// TwinCAT 3 PLC project Testlibrary
// Title: TestFramework
// Company: Hoox.Software
// Author: Patrick Dressel
// ProjectVersion: 2.2.6
// ProgramVersion: 3.1.4022.6
// libraries:
//   Tc2_Standard, * (Beckhoff Automation GmbH)
//   Tc2_System, * (Beckhoff Automation GmbH)
//   Tc2_Utilities, * (Beckhoff Automation GmbH)
//   Tc3_Module, * (Beckhoff Automation GmbH)
//   Base Interfaces,newest,System
// project tree:
//   Datatypes/ EResult_t.TcDUT, EAssertion_t.TcDUT (not stored), ERetCode_t.TcDUT (not stored), EState_t.TcDUT, IdHandle_t.TcDUT (not stored), ObjectId_t.TcDUT (not stored), SStatistic_t.TcDUT (not stored), STestcase_t.TcDUT, StringHandle_t.TcDUT (not stored), StrMessage_t.TcDUT (not stored), TestCaseHandle_t.TcDUT (not stored)
//   Datatypes/Report/ EExportState_t.TcDUT, EReportType_t.TcDUT (not stored), NameHandle_t.TcDUT (not stored), PathHandle_t.TcDUT (not stored), StrFileName_t.TcDUT (not stored), StrPathName_t.TcDUT (not stored), TestReportHandle_t.TcDUT (not stored), UBaseTypes_t.TcDUT (not stored), UTime_t.TcDUT (not stored)
//   GVLs/ GVL_Sample.TcGVL (excluded from build)
//   / GVL_Parameter.TcGVL, PlcTask.TcTTO
//   Source/Report/File/ FB_CoverageFile.TcPOU, FB_FileBase.TcPOU, FB_TestReportBase.TcPOU, FB_TextReport.TcPOU, IFileData_t.TcIO
//   Source/Report/Format/ EXmlFormat_t.TcDUT, FB_XmlTag.TcPOU, _CONCAT.TcPOU, _LEN.TcPOU
//   Source/Testlib/ FB_Assertion.TcPOU (not stored), PRG_TestLib.TcPOU
//   Source/Testsuite/ FB_Testsuite.TcPOU, ITestsuite_t.TcIO
//   Source/TestBase/ FB_TestBase.TcPOU (not stored), ITestBase_t.TcIO
//   Test/ FB_Test_Base.TcPOU, FB_Test_Base_Ptr.TcPOU, FB_Test_Base_Not.TcPOU, FB_Test_Base_Delay.TcPOU, PRG_Temp.TcPOU
// real-time tasks:
//   TASK PlcTask: cycle T#10ms, priority 20, ADS port 350

CONFIGURATION Testlibrary
    RESOURCE PLC ON TwinCAT3
        TASK PlcTask(INTERVAL := T#10ms, PRIORITY := 20);
        PROGRAM PRG_TestLib WITH PlcTask : PRG_TestLib;
        PROGRAM PRG_Temp WITH PlcTask : PRG_Temp;
    END_RESOURCE
END_CONFIGURATION

// ---- Datatypes/EResult_t.TcDUT
{attribute 'qualified_only'}
{attribute 'strict'}
TYPE EResult_t :
(
   eStateIdle,
	eStateSkipped,
	eStatePassed,
	eStateFailed,
	eStateFailedFatal
);
END_TYPE

// ---- Datatypes/EState_t.TcDUT
{attribute 'qualified_only'}
{attribute 'strict'}
TYPE EState_t :
(
	eStateInit,
	eStateIdle,
	eStatePrepare,
	eStateExecute,
	eStateCleanUp,
	eStateBuildUnitTestFile,
	eStateReady,
	eStateExport,
	eStateError,
	eStateLicenseError
);
END_TYPE

// ---- Datatypes/Report/EExportState_t.TcDUT
{attribute 'qualified_only'}
{attribute 'strict'}
TYPE EExportState_t :
(
	eExportIdle := 0,
	eExportOpen,
	eExportGetLine,
	eExportWrite,
	eExportClose,
	eExportError
);
END_TYPE

// ---- Datatypes/STestcase_t.TcDUT
TYPE STestcase_t :
STRUCT
	u32Passed 		: UDINT;
	u32Failed 		: UDINT;
	u32Time         : UDINT;
	eState          : EResult_t;
END_STRUCT
END_TYPE

// ---- Source/Report/Format/EXmlFormat_t.TcDUT
{attribute 'qualified_only'}
{attribute 'strict'}
TYPE EXmlFormat_t :
(
	ePlainXml := 0,
	eStructuredXml
);
END_TYPE

// ---- GVLs/GVL_Sample.TcGVL
{attribute 'qualified_only'}
VAR_GLOBAL
	// This File is only a simple Demo to show the usage of the Library
    // Using the Sccx-Script it can be generated by a build server like Jenkins

	// Report Instance 
	fb_TestReport : FB_TextReport;	
	
	// Register Testsuite
    // Testuite connects itself to PRG_TestLib
	fb_TestSuite1 : FB_Testsuite(i_strId 	:= 'TestSuite1', 	
								 i_strPath	:= 'Testframework\Testframework\UnitTest\');
	
	// Register Test in Testsuite1
    // Testcase connect itself to given Testsuite interface
    // set Execute to false to skip the test.
	fb_Test   : FB_Test_Base( i_strId 	 	    := 'TF1.1',
                              i_strClassName	:= 'FB_TestBase.TcPOU',
                              i_strPath 		:= 'Source',
                              i_iTestSuite 	    := fb_TestSuite1,
                              i_bExecute   	    := TRUE);
										
	fb_Test2   : FB_Test_Base( i_strId 	 	    := 'TF2.1',
                              i_strClassName	:= 'FB_TestBase.TcPOU',
                              i_strPath 		:= 'Source',
                              i_iTestSuite 	    := fb_TestSuite1,
                              i_bExecute   	    := TRUE);										
END_VAR

// ---- GVL_Parameter.TcGVL
{attribute 'qualified_only'}
VAR_GLOBAL CONSTANT
	strExportDirectory : STRING := 'C:\testresult\';
END_VAR

// ---- Source/Report/File/IFileData_t.TcIO
INTERFACE IFileData_t

METHOD getDataPtr : POINTER TO BYTE
END_METHOD

METHOD getSize : UDINT
VAR_INPUT
END_VAR
END_METHOD

END_INTERFACE

// ---- Source/Testsuite/ITestsuite_t.TcIO
INTERFACE ITestsuite_t

METHOD PUBLIC addTestcase : BOOL
VAR_INPUT
	i_iTestCase : ITestBase_t;
END_VAR
END_METHOD

METHOD execute : BOOL
VAR_INPUT
    i_bStart : BOOL;
END_VAR
END_METHOD

METHOD getFirstTestCase : ITestBase_t
VAR_INPUT
END_VAR
END_METHOD

METHOD getId : STRING
VAR_INPUT
END_VAR
END_METHOD

METHOD getNextTestCase : ITestBase_t
VAR_INPUT
END_VAR
END_METHOD

METHOD getPath : ObjectId_t
VAR_INPUT
END_VAR
END_METHOD

METHOD getResult : EResult_t
VAR_INPUT
END_VAR
END_METHOD

METHOD getState : EState_t
VAR_INPUT
END_VAR
END_METHOD

PROPERTY Result : SStatistic_t
GET
END_GET
END_PROPERTY

END_INTERFACE

// ---- Source/TestBase/ITestBase_t.TcIO
INTERFACE ITestBase_t

METHOD PUBLIC FINAL _cleanup : ERetCode_t
VAR_INPUT
END_VAR
END_METHOD

METHOD PUBLIC FINAL _execute : ERetCode_t
VAR_INPUT
END_VAR
END_METHOD

METHOD PUBLIC FINAL _prepare : ERetCode_t
VAR_INPUT
END_VAR
END_METHOD

METHOD getClassname : ObjectId_t
VAR_INPUT
END_VAR
END_METHOD

METHOD getId : ObjectId_t
VAR_INPUT
END_VAR
END_METHOD

METHOD getMessage : StrMessage_t
VAR_INPUT
END_VAR
END_METHOD

METHOD getPath : ObjectId_t
VAR_INPUT
END_VAR
END_METHOD

PROPERTY Result : STestcase_t
GET
END_GET
END_PROPERTY

END_INTERFACE

// ---- Source/Testlib/PRG_TestLib.TcPOU
(******************************************************************************
Baustein: PRG_TestLibrary
Spezifikation: doc/Spezifikation.pdf, Kap. x.y.z
-------------------------------------------------------------------------------
erstellt:
von:
Geändert:
von:
-------------------------------------------------------------------------------
Beschreibung
Dieser Baustein etnhält alle Testsuites und führt diese aus.

-------------------------------------------------------------------------------
Input
	i_bStart : mit positiver Flanke werden die registrierten Testsuites ausgeführt

Output
	o_eState  		: EState_t;
	o_eResult 		: EResult_t;
	o_sStatistic	: SStatistic_t;
******************************************************************************)
{attribute 'global_init_slot' := '41000'}
PROGRAM PRG_TestLib
VAR_INPUT
	i_bStart : BOOL;
END_VAR
VAR_OUTPUT
	o_eState  		: EState_t;
	o_eResult 		: EResult_t;
	o_sStatistic	: SStatistic_t;
END_VAR
VAR
	bHwStart AT %I* : BOOL;
	bHwBusy  AT %Q* : BOOL;
	bHwReady AT %Q* : BOOL;
	
	a_iTestSuite 	: ARRAY [0..255] OF ITestSuite_t;
	u16TestSuites 	: UINT;
	u16Index	  		: UINT;
	iActTestSuite 	: ITestSuite_t;
	pTestReport		: POINTER TO FB_TestReportBase;
	eRetCode 		: ERetCode_t;

	fbSystemTime 		: FB_LocalSystemTime;
	
	fbExportFolder		: FB_CreateDir;
	fbUnittest 			: FB_CoverageFile;
	u16ReportState  	: UINT;
	u16TestSuitIdx		: UINT;
	iTestCase  			: ITestBase_t;
	sTempResult     	: SStatistic_t;
	
	xmlTestsuites	  	: FB_XmlTag;
	xmlTestsuite	  	: FB_XmlTag;
	xmlTest	  			: FB_XmlTag;
	xmlTestResult		: FB_XmlTag;		
END_VAR
VAR CONSTANT 
	ADSERR_DEVICE_ACCESSDENIED : UDINT := 16#723;
	ADSERR_DEVICE_NOTFOUND     : UDINT := 16#70C;
	ADSERR_DEVICE_EXISTS     	: UDINT := 16#70F;
END_VAR


	fbSystemTime(bEnable := TRUE, dwCycle := 5);
			
	fbUnittest();

	CASE o_eState OF 
	
	EState_t.eStateInit:	
		
		IF checkExportFolder() THEN 
		   logInfo('Testlib V2.2.6 Ready');
			o_eState := EState_t.eStateIdle; 
		END_IF

	EState_t.eStateIdle:
	
		IF i_bStart = TRUE OR bHwStart = TRUE THEN
			logInfo('+++++++++++++ Testbeginn ++++++++++++++');
			o_eState := EState_t.eStatePrepare;
			bHwReady := FALSE;
		END_IF
	
	EState_t.eStatePrepare:
	
		bHwBusy := TRUE;
		
		o_eResult 	  					:= EResult_t.eStatePassed;
		o_sStatistic.u32Executed 	:= 0;
		o_sStatistic.u32TestCases	:= 0;
		o_sStatistic.u32Asserts  	:= 0;
		o_sStatistic.u32Passed   	:= 0;
		o_sStatistic.u32Failed	 	:= 0;	

		iActTestSuite := getFirstTestSuite();
		
		IF iActTestSuite      <> 0   THEN
			o_eState := EState_t.eStateExecute;
		ELSE
			o_eState := EState_t.eStateError;	
		END_IF
	
	EState_t.eStateExecute:
	
		iActTestSuite.execute(i_bStart := TRUE);
	
		IF iActTestSuite.getState() = EState_t.eStateReady THEN
			
			IF iActTestSuite.getResult() = EResult_t.eStateFailed THEN
				o_eResult := EResult_t.eStateFailed;
			END_IF
			
			iActTestSuite.execute(i_bStart := FALSE);
			sTempResult := iActTestSuite.Result;

			o_eState := EState_t.eStateCleanUp;

			o_sStatistic.u32Executed 	:= o_sStatistic.u32Executed  + sTempResult.u32Executed;
			o_sStatistic.u32TestCases	:= o_sStatistic.u32TestCases + sTempResult.u32TestCases; 
			o_sStatistic.u32Asserts  	:= o_sStatistic.u32Asserts   + sTempResult.u32Asserts;
			o_sStatistic.u32Passed   	:= o_sStatistic.u32Passed    + sTempResult.u32Passed;
			o_sStatistic.u32Failed	 	:= o_sStatistic.u32Failed    + sTempResult.u32Failed;
		END_IF
	
	EState_t.eStateCleanUp:
	
		IF iActTestSuite.getResult() = EResult_t.eStateFailedFatal THEN
			o_eResult := EResult_t.eStateFailedFatal;
			o_eState  := EState_t.eStateExport;
			logInfo('+++++++++++++ Fatal Error : Test Ende ++++++++++++++');
		ELSE
			
			iActTestSuite := getNextTestSuite();
						
			IF iActTestSuite <> 0 THEN
				o_eState := EState_t.eStateExecute;
			ELSE
				o_eState := EState_t.eStateBuildUnitTestFile;
				logInfo('+++++++++++++ Test Ende ++++++++++++++');
			END_IF		
			
		END_IF

	EState_t.eStateExport:

		IF createReport(EReporttype_t.eExternalReport) = ERetCode_t.eRetDone THEN
			o_eState := EState_t.eStateBuildUnitTestFile;
		END_IF;
		
	EState_t.eStateBuildUnitTestFile:

		IF createReportnew(EReporttype_t.eUnitTestReport) = ERetCode_t.eRetDone THEN
			o_eState := EState_t.eStateReady;
		END_IF;
		
	EState_t.eStateReady:

		bHwReady := TRUE;
		bHwBusy  := FALSE;
		IF i_bStart  = FALSE AND 
			bHwStart = FALSE THEN
			o_eState := EState_t.eStateIdle;
		END_IF		
		
	EState_t.eStateError,
	EState_t.eStateLicenseError:
	
		bHwBusy  := FALSE;
		o_eState := EState_t.eStateError;

	END_CASE

(******************************************************************************
Baustein: PRG_UnitTestLib.addTestReport
Spezifikation: doc/Spezifikation.pdf, Kap. x.y.z
-------------------------------------------------------------------------------
erstellt:
von:
Geändert:
von:
-------------------------------------------------------------------------------
Beschreibung
Diese Methode

-------------------------------------------------------------------------------
Input
i_pTestReport

Output
-
******************************************************************************)
{attribute 'hide'} 
METHOD PUBLIC addTestReport : BOOL
VAR_INPUT
	i_pTestReport : TestReportHandle_t;
END_VAR

	pTestReport := i_pTestReport;
END_METHOD

(******************************************************************************
Baustein: PRG_UnitTestLib.addTestSuite
Spezifikation: doc/Spezifikation.pdf, Kap. x.y.z
-------------------------------------------------------------------------------
erstellt:
von:
Geändert:
von:
-------------------------------------------------------------------------------
Beschreibung
Diese Methode

-------------------------------------------------------------------------------
Input
i_pTestSuite

Output
-
******************************************************************************)
{attribute 'hide'} 
METHOD PUBLIC addTestSuite : BOOL
VAR_INPUT
	i_iTestSuite : ITestSuite_t;
END_VAR
VAR
    sStatistic : SStatistic_t;
END_VAR

	addTestSuite := FALSE;

	IF 	i_iTestSuite  <> 0   AND 
		u16TestSuites <  255 THEN
		
		a_iTestSuite[u16TestSuites] := i_iTestSuite;
		sStatistic      := i_iTestSuite.Result;
		u16TestSuites   := u16TestSuites +1;
	
		o_sStatistic.u32TestSuites := o_sStatistic.u32TestSuites + 1;
		o_sStatistic.u32TestCases  := o_sStatistic.u32TestCases + sStatistic.u32TestCases;
		
		addTestSuite := TRUE;
	END_IF
END_METHOD

// 
// Lt. Infosys wird ADSERR_DEVICE_ACCESSDENIED zurückgegeben wenn der
// Ordner bereits existiert. Das reicht an der Stelle um zu wissen das 
// es soweit passt.
{attribute 'hide'} 
METHOD INTERNAL checkExportFolder : BOOL

	checkExportFolder := FALSE;
	
	fbExportFolder(sNetId 		:= '',
						sPathName 	:= GVL_Parameter.strExportDirectory,
						ePath 		:= E_OpenPath.PATH_GENERIC,
						bExecute 	:= TRUE,
						tTimeout 	:= T#5S);
						
	IF (fbExportFolder.bBusy  = FALSE) AND 
		(fbExportFolder.bError = FALSE OR 
			fbExportFolder.nErrId = ADSERR_DEVICE_ACCESSDENIED OR 
			fbExportFolder.nErrId = ADSERR_DEVICE_EXISTS 		OR 
			fbExportFolder.nErrId = ADSERR_DEVICE_NOTFOUND) THEN
		checkExportFolder := true;
	END_IF;
END_METHOD

{attribute 'hide'} 
METHOD PRIVATE createReport : ERetCode_t
VAR_INPUT
	i_eReporttype : EReportType_t;
END_VAR
VAR
	eRetcode    : ERetCode_t;
	u32Temp     : UDINT;
	sTestResult : STestcase_t;
	sStatistic  : SStatistic_t;
END_VAR

	createReport := ERetCode_t.eRetBusy;

	CASE u16ReportState OF

	0: 
		IF i_eReporttype = EReportType_t.eUnitTestReport THEN
			u16ReportState := 20;
		END_IF;

		IF i_eReporttype = EReportType_t.eExternalReport THEN
			u16ReportState := 100;
		END_IF;

// +++++++++++++++++++++++++++++++++++++++++++++++++++++++++++
//
// Export Unittest Ergebnisse
// 
// +++++++++++++++++++++++++++++++++++++++++++++++++++++++++++
	20:		

		eRetcode := fbUnitTest.open(GVL_Parameter.strExportDirectory, 'Unittest.xml');

		IF eRetcode = ERetCode_t.eRetDone THEN

			u16ReportState := 21;

		ELSIF eRetcode = ERetCode_t.eRetFailed THEN

			logError('createReport Unittest.xml : Datei nicht geöffnet');
			u16ReportState := 22;

		END_IF;	

	21:

		u16TestSuitIdx := 0;

		fbUnitTest.addString('<?xml version="1.0" ?>');
		fbUnitTest.addCrlf();

		iActTestSuite := getFirstTestSuite();
		fbUnitTest.addString('<testsuites>');
		fbUnitTest.addCrlf();

		WHILE (iActTestSuite <> 0) DO

            sStatistic := iActTestSuite.Result;
			u16TestSuitIdx := u16TestSuitIdx+1;

			fbUnitTest.addString('<testsuite');
			fbUnitTest.addString(' name="');
			fbUnitTest.addString(iActTestSuite.getId());
			fbUnitTest.addString('" tests="');			
			fbUnitTest.addValue(sStatistic.u32TestCases);
			fbUnitTest.addString('" disabled="');
            u32Temp := sStatistic.u32TestCases-sStatistic.u32Executed;
			fbUnitTest.addValue(u32Temp);
			fbUnitTest.addString('" errors="');
			fbUnitTest.addValue(u32Temp);
			fbUnitTest.addString('" failures="');
			fbUnitTest.addValue(sStatistic.u32Failed);
			fbUnitTest.addString('" hostname="');
			fbUnitTest.addString('" id="');
			fbUnitTest.addvalue(u16TestSuitIdx);
			fbUnitTest.addString('" package="');
			fbUnitTest.addString(iActTestSuite.getPath());
			fbUnitTest.addString('">');
			fbUnitTest.addCrlf();

			iTestCase := iActTestSuite.getFirstTestCase();

			WHILE (iTestCase <> 0) DO
        
                sTestResult := iTestCase.Result;

				fbUnitTest.addString('<testcase');
				fbUnitTest.addString(' name="');
				fbUnitTest.addString(iTestCase.getId());
				fbUnitTest.addString('" assertions="');
                u32Temp := sTestResult.u32Failed + sTestResult.u32Passed;
				fbUnitTest.addValue(u32Temp);
				fbUnitTest.addString('" classname="');
				fbUnitTest.addString(iTestCase.getPath());
                fbUnitTest.addString('.');
				fbUnitTest.addString(iTestCase.getClassName());
				fbUnitTest.addString('" time="');				
				fbUnitTest.addTimeMs(sTestResult.u32Time);
				fbUnitTest.addString('">');
				fbUnitTest.addCrlf();

				CASE sTestResult.eState OF

				EResult_t.eStatePassed :

					fbUnitTest.addString('<passed/>');

				EResult_t.eStateFailed, 
				EResult_t.eStateFailedFatal :
			
					fbUnitTest.addString('<failure');
					fbUnitTest.addString(' message="');
					fbUnitTest.addString(iTestCase.getMessage());
					fbUnitTest.addString('"/>');
					
				EResult_t.eStateSkipped:

					fbUnitTest.addString('<skipped/>');

				END_CASE;
				
				fbUnitTest.addCrlf();	

				fbUnitTest.addString('</testcase>');
				fbUnitTest.addCrlf();		

				iTestCase := iActTestSuite.getNextTestCase();
		
			END_WHILE

			fbUnitTest.addString('</testsuite>');
			fbUnitTest.addCrlf();	

			iActTestSuite := getNextTestSuite();

		END_WHILE

		fbUnitTest.addString('</testsuites>');
		fbUnitTest.addCrlf();

		u16ReportState := 22;

	22:
		IF fbUnitTest.o_bOpen  = TRUE AND 
		   fbUnitTest.o_bEmpty = TRUE THEN
			fbUnitTest.close();
		END_IF;

		IF fbUnitTest.o_bOpen  = FALSE THEN
			createReport 	:= ERetCode_t.eRetDone;
		END_IF;

// +++++++++++++++++++++++++++++++++++++++++++++++++++++++++++
//
//
// 
// +++++++++++++++++++++++++++++++++++++++++++++++++++++++++++
	100:

		IF pTestReport <> 0 THEN
			
			createReport := pTestReport^.create();		
			
		ELSE

			createReport := ERetCode_t.eRetDone;

		END_IF;

	ELSE
		createReport := ERetCode_t.eRetFailed;
	END_CASE;

	IF createReport = ERetCode_t.eRetDone THEN
		u16ReportState := 0;
	END_IF;
















(**)
END_METHOD

{attribute 'hide'} 
METHOD PRIVATE createReportNew : ERetCode_t
VAR_INPUT
	i_eReporttype : EReportType_t;
END_VAR
VAR
	eRetcode    : ERetCode_t;
	u32Temp     : UDINT;
	sTestResult : STestcase_t;
	sStatistic  : SStatistic_t;
	

END_VAR

	createReportNew := ERetCode_t.eRetBusy;

	CASE u16ReportState OF

	0: 
		IF i_eReporttype = EReportType_t.eUnitTestReport THEN
			u16ReportState := 20;
		END_IF;
		
// +++++++++++++++++++++++++++++++++++++++++++++++++++++++++++
//
// Export Unittest Ergebnisse
// 
// +++++++++++++++++++++++++++++++++++++++++++++++++++++++++++
	20:		

		eRetcode := fbUnitTest.open(GVL_Parameter.strExportDirectory, 'Unittest.xml');

		IF eRetcode = ERetCode_t.eRetDone THEN

			u16ReportState := 21;

		ELSIF eRetcode = ERetCode_t.eRetFailed THEN

			logError('createReport Unittest.xml : Datei nicht geöffnet');
			u16ReportState := 22;

		END_IF;	

	21:

		u16TestSuitIdx := 0;

		fbUnitTest.addString('<?xml version="1.0" ?>');
		fbUnitTest.addCrlf();

		xmlTestsuites.create('testsuites')
						 .setFormat(EXmlFormat_t.eStructuredXml)
						 .close();	
		
		iActTestSuite := getFirstTestSuite();

		WHILE (iActTestSuite <> 0) DO

         sStatistic	   := iActTestSuite.Result;
			u16TestSuitIdx := u16TestSuitIdx+1;

			xmlTestsuite.create('testsuite')
							.setFormat(EXmlFormat_t.eStructuredXml)
							.AddAttribute('name', 		iActTestSuite.getId())
							.AddAttribute('tests', 		UDINT_TO_STRING(sStatistic.u32TestCases))
							.AddAttribute('disabled', 	UDINT_TO_STRING(sStatistic.u32TestCases-sStatistic.u32Executed))
							.AddAttribute('errors', 	UDINT_TO_STRING(0))
							.AddAttribute('failures', 	UDINT_TO_STRING(sStatistic.u32Failed))
							.AddAttribute('hostname', 	'')
							.AddAttribute('id', 			UINT_TO_STRING(u16TestSuitIdx))
							.AddAttribute('package', 	iActTestSuite.getPath())
							.close();

			iTestCase := iActTestSuite.getFirstTestCase();

			WHILE (iTestCase <> 0) DO
        
            sTestResult := iTestCase.Result;
				
				xmlTest.create('testcase')			
						.setFormat(EXmlFormat_t.eStructuredXml)
						.AddAttribute('name', 			iTestCase.getId())
						.AddAttribute('assertions', 	UDINT_TO_STRING(sTestResult.u32Failed + sTestResult.u32Passed))
						.AddAttribute('classname', 	iTestCase.getClassName())
						.AddAttribute('time', 			UDINT_TO_STRING(sTestResult.u32Time))
						.close();

				CASE sTestResult.eState OF

				EResult_t.eStatePassed :

					xmlTestResult.create('passed')
									 .setFormat(EXmlFormat_t.eStructuredXml)
								 	 .close();

				EResult_t.eStateFailed, 
				EResult_t.eStateFailedFatal :
			
					xmlTestResult.create('failure')
									 .setFormat(EXmlFormat_t.eStructuredXml)
									 .AddAttribute('message', iTestCase.getMessage())
									 .close();
					
				EResult_t.eStateSkipped:

					xmlTestResult.create('skipped')
									 .setFormat(EXmlFormat_t.eStructuredXml)
								 	 .close();


				END_CASE;
				
				xmlTest.AddTag(xmlTestResult);				 
				xmlTestsuite.AddTag(xmlTest);

				iTestCase := iActTestSuite.getNextTestCase();
		
			END_WHILE

			xmlTestsuites.AddTag(xmlTestsuite);
						
			iActTestSuite := getNextTestSuite();

		END_WHILE
		
		fbUnitTest.addObject(xmlTestsuites);

		u16ReportState := 22;

	22:
		IF fbUnitTest.o_bOpen  = TRUE AND 
		   fbUnitTest.o_bEmpty = TRUE THEN
			fbUnitTest.close();
		END_IF;

		IF fbUnitTest.o_bOpen  = FALSE THEN
			createReportNew 	:= ERetCode_t.eRetDone;
		END_IF;

	ELSE
		createReportNew := ERetCode_t.eRetFailed;
	END_CASE;

	IF createReportNew = ERetCode_t.eRetDone THEN
		u16ReportState := 0;
	END_IF;
















(**)
END_METHOD

(******************************************************************************
Baustein: PRG_UnitTestLib.getFirstTestSuite
Spezifikation: doc/Spezifikation.pdf, Kap. x.y.z
-------------------------------------------------------------------------------
erstellt:
von:
Geändert:
von:
-------------------------------------------------------------------------------
Beschreibung
Diese Methode

-------------------------------------------------------------------------------
Input
-

Output
-
******************************************************************************)
{attribute 'hide'} 
METHOD PRIVATE getFirstTestSuite : ITestSuite_t
VAR_INPUT
END_VAR

	u16Index := 0;
	getFirstTestSuite := a_iTestSuite[0];
END_METHOD

(******************************************************************************
Baustein: PRG_UnitTestLib.getNextTestSuite
Spezifikation: doc/Spezifikation.pdf, Kap. x.y.z
-------------------------------------------------------------------------------
erstellt:
von:
Geändert:
von:
-------------------------------------------------------------------------------
Beschreibung
Diese Methode

-------------------------------------------------------------------------------
Input
-

Output
-
******************************************************************************)
{attribute 'hide'} 
METHOD PRIVATE getNextTestSuite : ITestSuite_t
VAR_INPUT
END_VAR

	getNextTestSuite := 0;
	u16Index 		 := u16Index + 1;

	IF u16Index < u16TestSuites THEN
		getNextTestSuite := a_iTestSuite[u16Index];
	END_IF;
END_METHOD

(******************************************************************************
Baustein: PRG_UnitTestLib.getTime
Spezifikation: doc/Spezifikation.pdf, Kap. x.y.z
-------------------------------------------------------------------------------
erstellt:
von:
Geändert:
von:
-------------------------------------------------------------------------------
Beschreibung
Diese Methode

-------------------------------------------------------------------------------
Input
-

Output
-
******************************************************************************)
{attribute 'hide'} 
METHOD getTime : TimeStruct
VAR_INPUT
END_VAR
VAR
END_VAR

	getTime := fbSystemTime.systemTime;
END_METHOD

(******************************************************************************
Baustein: PRG_UnitTestLib.logError
Spezifikation: doc/Spezifikation.pdf, Kap. x.y.z
-------------------------------------------------------------------------------
erstellt:
von:
Geändert:
von:
-------------------------------------------------------------------------------
Beschreibung
Diese Methode

-------------------------------------------------------------------------------
Input
i_strMessage

Output
-
******************************************************************************)
{attribute 'hide'} 
METHOD PROTECTED logError : BOOL
VAR_INPUT
	i_strMessage : StrMessage_t;
END_VAR

	ADSLOGSTR(msgCtrlMask 	:= ADSLOG_MSGTYPE_ERROR , 
			  msgFmtStr 	:= i_strMessage, 
			  strArg 		:= '');
END_METHOD

(******************************************************************************
Baustein: PRG_UnitTestLib.logInfo
Spezifikation: doc/Spezifikation.pdf, Kap. x.y.z
-------------------------------------------------------------------------------
erstellt:
von:
Geändert:
von:
-------------------------------------------------------------------------------
Beschreibung
Diese Methode

-------------------------------------------------------------------------------
Input
i_strMessage

Output
-
******************************************************************************)
{attribute 'hide'} 
METHOD PUBLIC logInfo : BOOL
VAR_INPUT
	i_strMessage : StrMessage_t;
END_VAR

	ADSLOGSTR(msgCtrlMask 	:= ADSLOG_MSGTYPE_HINT , 
			  msgFmtStr 	:= i_strMessage, 
			  strArg 		:= '');
END_METHOD

END_PROGRAM

// ---- Source/Report/File/FB_TestReportBase.TcPOU
(******************************************************************************
Baustein: FB_TestReportBase
Spezifikation: doc/Spezifikation.pdf, Kap. x.y.z
-------------------------------------------------------------------------------
erstellt:
von:
Geändert:
von:
-------------------------------------------------------------------------------
Beschreibung
Dieser Baustein enthält alle zugeordneten Testfälle. Ein Testfall
ist ein abgeleiteter Baustein (FB) von FB_TestBase.

-------------------------------------------------------------------------------
Input
-

Output
-
******************************************************************************)
FUNCTION_BLOCK FB_TestReportBase
VAR_INPUT
END_VAR
VAR_OUTPUT
END_VAR
VAR
	strBuffer   : STRING(255);
	fbOpen      : FB_FileOpen;
	fbClose     : FB_FileClose;
	fbWrite	    : FB_FileWrite;
	strFileName : StrFileName_t;
	strFilePath : StrPathName_t;
	
	eState 		: EExportState_t;
	u32Line     : UDINT;
	
	sStatistic  : SStatistic_t;

	trgOpen 		: F_TRIG;
	trgWrite 	: F_TRIG;
	trgClose 	: F_TRIG;
END_VAR

(******************************************************************************
Baustein: FB_TestReportBase.addCrlf
Spezifikation: doc/Spezifikation.pdf, Kap. x.y.z
-------------------------------------------------------------------------------
erstellt:
von:
Geändert:
von:
-------------------------------------------------------------------------------
Beschreibung


-------------------------------------------------------------------------------
Input
-

Output
-
******************************************************************************)
METHOD PROTECTED addCrlf : BOOL
VAR_INPUT
END_VAR
VAR
END_VAR
   
	strBuffer := CONCAT(strBuffer, '$R$N');
END_METHOD

(******************************************************************************
Baustein: FB_TestReportBase.addDate
Spezifikation: doc/Spezifikation.pdf, Kap. x.y.z
-------------------------------------------------------------------------------
erstellt:
von:
Geändert:
von:
-------------------------------------------------------------------------------
Beschreibung

-------------------------------------------------------------------------------
Input
	i_sDate : TIMESTRUCT;

Output
-
******************************************************************************)
METHOD PROTECTED addDate : ERetCode_t
VAR_INPUT
	i_sDate : TIMESTRUCT;
END_VAR

	addDate := ERetcode_t.eRetDone;
	
	addValue(i_sDate.wDay);
	addString('.');
	addValue(i_sDate.wMonth);
	addString('.');
	addValue(i_sDate.wYear);
	addString(' ');
END_METHOD

(******************************************************************************
Baustein: FB_TestReportBase.addString
Spezifikation: doc/Spezifikation.pdf, Kap. x.y.z
-------------------------------------------------------------------------------
erstellt:
von:
Geändert:
von:
-------------------------------------------------------------------------------
Beschreibung

-------------------------------------------------------------------------------
Input
	i_strData : STRING(255);

Output
-
******************************************************************************)
METHOD PROTECTED addString : ERetCode_t
VAR_INPUT
	i_strData : STRING(255);
END_VAR

	strBuffer :=  concat(strBuffer, i_strData);

	addString := ERetcode_t.eRetDone;
END_METHOD

(******************************************************************************
Baustein: FB_TestReportBase.addTime
Spezifikation: doc/Spezifikation.pdf, Kap. x.y.z
-------------------------------------------------------------------------------
erstellt:
von:
Geändert:
von:
-------------------------------------------------------------------------------
Beschreibung

-------------------------------------------------------------------------------
Input
	i_sTime : TIMESTRUCT;

Output
-
******************************************************************************)
METHOD PROTECTED addTime : ERetCode_t
VAR_INPUT
	i_sTime : TIMESTRUCT;
END_VAR

	addTime := ERetcode_t.eRetDone;
	
   	addValue(i_sTime.wHour);
   	addString('.');
   	addValue(i_sTime.wMinute);
  	addString('.');
   	addValue(i_sTime.wSecond);
   	addString(' ');
END_METHOD

(******************************************************************************
Baustein: FB_TestReportBase.addValue
Spezifikation: doc/Spezifikation.pdf, Kap. x.y.z
-------------------------------------------------------------------------------
erstellt:
von:
Geändert:
von:
-------------------------------------------------------------------------------
Beschreibung

-------------------------------------------------------------------------------
Input
	i_anyValue : ANY;

Output
-
******************************************************************************)
METHOD PROTECTED addValue : ERetCode_t
VAR_INPUT
	i_anyValue : ANY;
END_VAR
VAR
	uValue : UBaseTypes_t;
END_VAR

	addValue  := ERetcode_t.eRetDone;
	
	IF i_anyValue.pValue = 0 THEN
		addValue  := ERetcode_t.eRetFailed;
		RETURN;
	END_IF

	MEMCPY(ADR(uValue),i_anyValue.pValue, TO_UDINT(i_anyValue.diSize)); 

	CASE i_anyValue.TypeClass OF

	__SYSTEM.Type_Class.TYPE_SINT:

		addString(SINT_TO_STRING(uValue.s8Value));

	//__SYSTEM.Type_Class.TYPE_BYTE:
	__SYSTEM.Type_Class.TYPE_USINT:

		addString(USINT_TO_STRING(uValue.u8Value));

	__SYSTEM.Type_Class.TYPE_INT:

		addString(INT_TO_STRING(uValue.s16Value));

	__SYSTEM.Type_Class.TYPE_DINT:

		addString(DINT_TO_STRING(uValue.s32Value));

	__SYSTEM.Type_Class.TYPE_UINT:

		addString(UINT_TO_STRING(uValue.u16Value));

	__SYSTEM.Type_Class.TYPE_UDINT:

		addString(UDINT_TO_STRING(uValue.u32Value));

	__SYSTEM.Type_Class.TYPE_WORD:

		addString(WORD_TO_STRING(uValue.w16Value));

	__SYSTEM.Type_Class.TYPE_DWORD:

		addString(DWORD_TO_STRING(uValue.w32Value));

	ELSE
		ADSLOGSTR(msgCtrlMask 	:= ADSLOG_MSGTYPE_ERROR , 
				  msgFmtStr 	:= 'TestReportBase.AddValue - Unbekannter Datentyp!', 
				  strArg 		:= '');
	END_CASE;
END_METHOD

(******************************************************************************
Baustein: FB_TestReportBase.BuildFile
Spezifikation: doc/Spezifikation.pdf, Kap. x.y.z
-------------------------------------------------------------------------------
erstellt:
von:
Geändert:
von:
-------------------------------------------------------------------------------
Beschreibung
Diese Methode muss vom ableitenden Baustein überschrieben werden und
wird von der Basisklasse aus aufgerufen wenn der Report erstellt werden
soll.

-------------------------------------------------------------------------------
Input
-

Output
-
******************************************************************************)
METHOD PROTECTED BuildFile : ERetCode_t
VAR_INPUT
	i_u32Line : UDINT;
END_VAR
END_METHOD

(******************************************************************************
Baustein: FB_TestReportBase.clearBuffer
Spezifikation: doc/Spezifikation.pdf, Kap. x.y.z
-------------------------------------------------------------------------------
erstellt:
von:
Geändert:
von:
-------------------------------------------------------------------------------
Beschreibung

-------------------------------------------------------------------------------
Input
-

Output
-
******************************************************************************)
METHOD PROTECTED clearBuffer : ERetCode_t
VAR_INPUT
END_VAR

	clearBuffer := ERetCode_t.eRetDone;
	
	strBuffer := '';
END_METHOD

(******************************************************************************
Baustein: FB_TestReportBase.Close
Spezifikation: doc/Spezifikation.pdf, Kap. x.y.z
-------------------------------------------------------------------------------
erstellt:
von:
Geändert:
von:
-------------------------------------------------------------------------------
Beschreibung


-------------------------------------------------------------------------------
Input
-

Output
-
******************************************************************************)
METHOD PROTECTED Close : ERetCode_t
VAR_INPUT
END_VAR

	Close := ERetCode_t.eRetFailed;
	
	fbClose.hFile 		:= fbOpen.hFile;
	fbClose.bExecute 	:= TRUE; 

	IF trgClose.Q = TRUE THEN
		Close := ERetCode_t.eRetDone;
		fbClose.bExecute  := FALSE;		
	ELSE	
		Close := ERetCode_t.eRetBusy;
	END_IF;	
	
	IF fbClose.bError = TRUE THEN
		Close := eRetCode_t.eRetFailed;
	END_IF;
END_METHOD

(******************************************************************************
Baustein: FB_TestReportBase.create
Spezifikation: doc/Spezifikation.pdf, Kap. x.y.z
-------------------------------------------------------------------------------
erstellt:
von:
Geändert:
von:
-------------------------------------------------------------------------------
Beschreibung


-------------------------------------------------------------------------------
Input
-

Output
-
******************************************************************************)
METHOD PUBLIC create : ERetCode_t;
VAR_INPUT
END_VAR
VAR
	eRetCode : ERetCode_t;
END_VAR

	create := ERetCode_t.eRetBusy;

	fbOpen();
	fbWrite();
	fbClose();

	trgOpen(CLK := fbOpen.bBusy);
	trgWrite(CLK := fbWrite.bBusy);
	trgClose(CLK := fbClose.bBusy);
	
	CASE eState OF
	
	EExportState_t.eExportIdle:
	
		eState := EExportState_t.eExportOpen;
	
	EExportState_t.eExportOpen:
	
		eRetCode 	:= Open();
		u32Line  	:= 0;
		sStatistic 	:= PRG_TestLib.o_sStatistic;

		IF eRetCode = ERetCode_t.eRetDone THEN
			eState := EExportState_t.eExportGetLine;
		ELSIF eRetCode = ERetCode_t.eRetFailed THEN
			eState := EExportState_t.eExportError;
		END_IF;

	EExportState_t.eExportGetLine:

		eRetCode := BuildFile(u32Line);

		IF eRetCode = ERetCode_t.eRetDone THEN
			eState := EExportState_t.eExportClose;
		ELSIF eRetCode = ERetCode_t.eRetFailed THEN
			eState := EExportState_t.eExportError;
		ELSE
			addCrlf();
			eState := EExportState_t.eExportWrite;
		END_IF;

	EExportState_t.eExportWrite:
	
		IF writeBuffer() =  ERetCode_t.eRetDone THEN
			clearBuffer();	
			u32Line := u32Line + 1;
			eState  := EExportState_t.eExportGetLine;
		END_IF;		
	
	EExportState_t.eExportClose:
	
		eRetCode := Close();
		
		IF eRetCode = ERetCode_t.eRetDone THEN
			eState     := EExportState_t.eExportIdle;
			create	   := ERetCode_t.eRetDone;
			reset();
		ELSIF eRetCode = ERetCode_t.eRetFailed THEN
			eState := EExportState_t.eExportError;
		end_if;
	
	EExportState_t.eExportError:
	
		create := ERetCode_t.eRetFailed;
	
	end_case;
END_METHOD

(******************************************************************************
Baustein: FB_TestReportBase.FB_Init
Spezifikation: doc/Spezifikation.pdf, Kap. x.y.z
-------------------------------------------------------------------------------
erstellt:
von:
Geändert:
von:
-------------------------------------------------------------------------------
Beschreibung


-------------------------------------------------------------------------------
Input
-

Output
-
******************************************************************************)
METHOD FB_init : BOOL
VAR_INPUT
	bInitRetains : BOOL; // if TRUE, the retain variables are initialized (warm start / cold start)
	bInCopyCode : BOOL;  // if TRUE, the instance afterwards gets moved into the copy code (online change)
END_VAR

	PRG_TestLib.addTestReport(this);
END_METHOD

(******************************************************************************
Baustein: FB_TestReportBase.getFileName
Spezifikation: doc/Spezifikation.pdf, Kap. x.y.z
-------------------------------------------------------------------------------
erstellt:
von:
Geändert:
von:
-------------------------------------------------------------------------------
Beschreibung
Diese Methode muss vom ableitenden Baustein überschrieben werden und
wird von der Basisklasse aus aufgerufen wenn der Report erstellt werden
soll.

-------------------------------------------------------------------------------
Input
	i_pFileName : NameHandle_t;
	i_pPath		: PathHandle_t;

Output
-
******************************************************************************)
METHOD PROTECTED getFileName : ERetCode_t
VAR_INPUT
	i_pFileName : NameHandle_t;
	i_pPath		: PathHandle_t;
END_VAR
END_METHOD

(******************************************************************************
Baustein: FB_TestReportBase.getTime
Spezifikation: doc/Spezifikation.pdf, Kap. x.y.z
-------------------------------------------------------------------------------
erstellt:
von:
Geändert:
von:
-------------------------------------------------------------------------------
Beschreibung


-------------------------------------------------------------------------------
Input
-

Output
-
******************************************************************************)
METHOD PROTECTED getTime : TimeStruct
VAR_INPUT
END_VAR
VAR
END_VAR

	getTime := PRG_TestLib.getTime();
END_METHOD

(******************************************************************************
Baustein: FB_TestReportBase.Open
Spezifikation: doc/Spezifikation.pdf, Kap. x.y.z
-------------------------------------------------------------------------------
erstellt:
von:
Geändert:
von:
-------------------------------------------------------------------------------
Beschreibung


-------------------------------------------------------------------------------
Input
-

Output
-
******************************************************************************)
METHOD PROTECTED open : ERetCode_t
VAR_INPUT
END_VAR

	open := ERetCode_t.eRetFailed;

	getFileName(ADR(strFileName), ADR(strFilePath));
	
	fbOpen.sPathName := CONCAT(strFilePath, strFileName);
	fbOpen.nMode 	 := FOPEN_MODEWRITE OR FOPEN_MODEBINARY;	
	fbOpen.bExecute  := TRUE;
			
	IF trgOpen.Q = TRUE THEN
		open := ERetCode_t.eRetDone;
		fbOpen.bExecute  := FALSE;		
	ELSE	
		open := ERetCode_t.eRetBusy;
	END_IF;	
	
	IF fbOpen.bError = TRUE THEN
		open := eRetCode_t.eRetFailed;
	END_IF;
END_METHOD

(******************************************************************************
Baustein: FB_TestReportBase.reset
Spezifikation: doc/Spezifikation.pdf, Kap. x.y.z
-------------------------------------------------------------------------------
erstellt:
von:
Geändert:
von:
-------------------------------------------------------------------------------
Beschreibung


-------------------------------------------------------------------------------
Input
-

Output
-
******************************************************************************)
METHOD PUBLIC reset : BOOL
VAR_INPUT
END_VAR

	IF fbOpen.hFile <> 0 THEN
		close();
	END_IF
	
	clearBuffer();

	fbOpen(sPathName := '', bExecute := FALSE);
	
	fbWrite(bExecute := FALSE);
	
	fbClose(bExecute := FALSE);
	
	eState := EExportState_t.eExportIdle;
END_METHOD

(******************************************************************************
Baustein: FB_TestReportBase.writeBuffer
Spezifikation: doc/Spezifikation.pdf, Kap. x.y.z
-------------------------------------------------------------------------------
erstellt:
von:
Geändert:
von:
-------------------------------------------------------------------------------
Beschreibung


-------------------------------------------------------------------------------
Input
-

Output
-
******************************************************************************)
METHOD PROTECTED writeBuffer : ERetCode_t
VAR_INPUT
END_VAR
VAR
	u32Len : UDINT;
END_VAR

	writeBuffer := eRetCode_t.eRetBusy;
	
	IF LEN(strBuffer) <= 0 THEN
		RETURN;
	END_IF
	
	u32Len := TO_UDINT(LEN(strBuffer)); 
	
	writeBuffer := writeData(i_pData := ADR(strBuffer), u32Size := u32Len);
END_METHOD

(******************************************************************************
Baustein: FB_TestReportBase.writeData
Spezifikation: doc/Spezifikation.pdf, Kap. x.y.z
-------------------------------------------------------------------------------
erstellt:
von:
Geändert:
von:
-------------------------------------------------------------------------------
Beschreibung


-------------------------------------------------------------------------------
Input
	i_pData : POINTER TO BYTE;
	u32Size : UDINT;
	
Output
-
******************************************************************************)
METHOD PROTECTED writeData : ERetCode_t
VAR_INPUT
	i_pData : POINTER TO BYTE;
	u32Size : UDINT;
END_VAR

	writeData := ERetCode_t.eRetFailed;
	
	IF u32Size = 0 OR i_pData = 0 THEN
		RETURN;
	END_IF
	
	fbWrite.pWriteBuff 	:= i_pData; 
	fbWrite.cbWriteLen 	:= u32Size; 
	fbWrite.hFile 		:= fbOpen.hFile; 
	fbWrite.bExecute 	:= TRUE;
			
	IF trgWrite.Q = TRUE THEN
		writeData := ERetCode_t.eRetDone;
		fbWrite.bExecute 	:= FALSE;			
	ELSE	
		writeData := ERetCode_t.eRetBusy;
	END_IF;	

	IF fbWrite.bError = TRUE THEN
		writeData := eRetCode_t.eRetFailed;
	END_IF;
END_METHOD

END_FUNCTION_BLOCK

// ---- Source/Report/File/FB_CoverageFile.TcPOU
FUNCTION_BLOCK FB_CoverageFile EXTENDS FB_FileBase


	writeBuffer();

	SUPER^();

END_FUNCTION_BLOCK

// ---- Source/Report/File/FB_FileBase.TcPOU
(******************************************************************************
Baustein: FB_TestReportBase
Spezifikation: doc/Spezifikation.pdf, Kap. x.y.z
-------------------------------------------------------------------------------
erstellt:
von:
Geändert:
von:
-------------------------------------------------------------------------------
Beschreibung
Dieser Baustein enthält alle zugeordneten Testfälle. Ein Testfall
ist ein abgeleiteter Baustein (FB) von FB_TestBase.

-------------------------------------------------------------------------------
Input
-

Output
-
******************************************************************************)
FUNCTION_BLOCK FB_FileBase
VAR_INPUT
END_VAR
VAR_OUTPUT
	o_bOpen 	: BOOL;
	o_bError 	: BOOL;
	o_bEmpty 	: BOOL;
END_VAR
VAR
	Buffer      : ARRAY[0..16384] OF BYTE;
	u32RdIdx    : UDINT;
	u32WrIdx    : UDINT;
	u32MaxIdx   : UDINT := 16384;
	
	fbOpen      : FB_FileOpen;
	fbClose     : FB_FileClose;
	fbWrite	   : FB_FileWrite;
	strFileName : StrFileName_t;
	strFilePath : StrPathName_t;
	
	eState 		: EExportState_t;
	u32Line     : UDINT;
	
	sStatistic  : SStatistic_t;

	trgOpen 	   : F_TRIG;
	trgWrite 	: F_TRIG;
	trgClose 	: F_TRIG;
END_VAR


	fbOpen();
	fbWrite();
	fbClose();
	
	trgOpen(CLK := fbOpen.bBusy);
	IF trgOpen.Q = TRUE THEN
		fbOpen.bExecute := FALSE;
	END_IF;

	trgWrite(CLK := fbWrite.bBusy);
	IF trgWrite.Q = TRUE THEN
		fbWrite.bExecute := FALSE;
	END_IF;

	trgClose(CLK := fbClose.bBusy);
	IF trgClose.Q = TRUE THEN
		fbClose.bExecute := FALSE;
	END_IF;

	o_bEmpty := (u32WrIdx = u32RdIdx);

(******************************************************************************
Baustein: FB_TestReportBase.addCrlf
Spezifikation: doc/Spezifikation.pdf, Kap. x.y.z
-------------------------------------------------------------------------------
erstellt:
von:
Geändert:
von:
-------------------------------------------------------------------------------
Beschreibung


-------------------------------------------------------------------------------
Input
-

Output
-
******************************************************************************)
METHOD PUBLIC addCrlf : ERetCode_t
VAR_INPUT
END_VAR
VAR
	strTemp : string := '$R$N';
END_VAR

	addData(adr(strTemp), 2);
	
	addCrlf := ERetCode_t.eRetDone;
END_METHOD

METHOD PRIVATE addData : BOOL
VAR_INPUT
	pData   : POINTER TO BYTE;
	u32Size : UDINT;
END_VAR
VAR
	u32Part1 : UDINT;
	u32Part2 : UDINT;
END_VAR

	IF u32WrIdx + u32Size <= u32MaxIdx THEN
		MemCpy(ADR(buffer)+u32WrIdx, pData, u32Size);
		u32WrIdx := u32WrIdx + u32Size;
	ELSE
		// buffer bis maximum beschreiben und den rest
		// vorne einfügen
		u32Part1 := u32MaxIdx-u32WrIdx;
		u32Part2 := u32Size - u32Part1;

		MemCpy(ADR(buffer) + u32WrIdx, pData, u32Part1);
		
		MemCpy(ADR(buffer), pData+u32Part1, u32Part2);
		// Schreibindex ist dann die Restgröße in Byte
		u32WrIdx := u32Part2;
	END_IF
END_METHOD

METHOD PUBLIC addObject : BOOL
VAR_INPUT
	iObject : IFileData_t;
END_VAR

	addData(iObject.getDataPtr(), iObject.getSize());
END_METHOD

(******************************************************************************
Baustein: FB_TestReportBase.addString
Spezifikation: doc/Spezifikation.pdf, Kap. x.y.z
-------------------------------------------------------------------------------
erstellt:
von:
Geändert:
von:
-------------------------------------------------------------------------------
Beschreibung

-------------------------------------------------------------------------------
Input
	i_strData : STRING(255);

Output
-
******************************************************************************)
METHOD PUBLIC addString : ERetCode_t
VAR_INPUT
	i_strData : STRING(1024);
END_VAR

	addData(ADR(i_strData), len(i_strData));
	
	addString := ERetcode_t.eRetDone;
END_METHOD

METHOD PUBLIC addTimeMs : ERetCode_t
VAR_INPUT
	i_u32Value : UDINT;
END_VAR
VAR
	strTemp  : STRING;
	s16Len   : INT;
END_VAR


		strTemp := UDINT_TO_STRING(i_u32Value);
		s16Len  := len(strTemp);

		IF s16Len < 4 THEN

			WHILE s16Len < 3 DO
				strTemp := concat('0', strTemp);
				s16Len  := len(strTemp);
			END_WHILE

			strTemp := concat('.', strTemp);
			strTemp := concat('0', strTemp);

		END_IF;

		PRG_TestLib.logInfo(concat('addTimeMs : ' , strTemp));

		addString(strTemp);
END_METHOD

(******************************************************************************
Baustein: FB_TestReportBase.addValue
Spezifikation: doc/Spezifikation.pdf, Kap. x.y.z
-------------------------------------------------------------------------------
erstellt:
von:
Geändert:
von:
-------------------------------------------------------------------------------
Beschreibung

-------------------------------------------------------------------------------
Input
	i_anyValue : ANY;

Output
-
******************************************************************************)
METHOD PUBLIC addValue : ERetCode_t
VAR_INPUT
	i_anyValue : ANY;
END_VAR
VAR
	uValue : UBaseTypes_t;
END_VAR

	addValue  := ERetcode_t.eRetDone;
	
	IF i_anyValue.pValue = 0 THEN
		addValue  := ERetcode_t.eRetFailed;
		RETURN;
	END_IF

	MEMCPY(ADR(uValue),i_anyValue.pValue, TO_UDINT(i_anyValue.diSize)); 

	CASE i_anyValue.TypeClass OF

	__SYSTEM.Type_Class.TYPE_SINT:

		addString(SINT_TO_STRING(uValue.s8Value));

	__SYSTEM.Type_Class.TYPE_USINT:

		addString(USINT_TO_STRING(uValue.u8Value));

	__SYSTEM.Type_Class.TYPE_INT:

		addString(INT_TO_STRING(uValue.s16Value));

	__SYSTEM.Type_Class.TYPE_DINT:

		addString(DINT_TO_STRING(uValue.s32Value));

	__SYSTEM.Type_Class.TYPE_UINT:

		addString(UINT_TO_STRING(uValue.u16Value));

	__SYSTEM.Type_Class.TYPE_UDINT:

		addString(UDINT_TO_STRING(uValue.u32Value));

	__SYSTEM.Type_Class.TYPE_WORD:

		addString(WORD_TO_STRING(uValue.w16Value));

	__SYSTEM.Type_Class.TYPE_DWORD:

		addString(DWORD_TO_STRING(uValue.w32Value));

	__SYSTEM.Type_Class.TYPE_BYTE:

		addString(BYTE_TO_STRING(uValue.u8Value));

	__SYSTEM.Type_Class.TYPE_BOOL:
		
		IF (uValue.bValue = TRUE) THEN
			addString('TRUE');
		ELSE
			addString('FALSE');
		END_IF;

	__SYSTEM.Type_Class.TYPE_REAL:
		
		addString(REAL_TO_STRING(uValue.r32Value));
	
	ELSE
		ADSLOGSTR(msgCtrlMask 	:= ADSLOG_MSGTYPE_ERROR , 
				  msgFmtStr 	:= 'TestReportBase.AddValue - Unbekannter Datentyp!', 
				  strArg 		:= '');
	END_CASE;
END_METHOD

(******************************************************************************
Baustein: FB_TestReportBase.clearBuffer
Spezifikation: doc/Spezifikation.pdf, Kap. x.y.z
-------------------------------------------------------------------------------
erstellt:
von:
Geändert:
von:
-------------------------------------------------------------------------------
Beschreibung

-------------------------------------------------------------------------------
Input
-

Output
-
******************************************************************************)
METHOD PUBLIC clearBuffer : ERetCode_t
VAR_INPUT
END_VAR

	clearBuffer := ERetCode_t.eRetDone;
	
	MemSet(ADR(buffer), 0, SIZEOF(buffer));
	
	u32WrIdx := u32RdIdx := 0;
END_METHOD

(******************************************************************************
Baustein: FB_TestReportBase.Close
Spezifikation: doc/Spezifikation.pdf, Kap. x.y.z
-------------------------------------------------------------------------------
erstellt:
von:
Geändert:
von:
-------------------------------------------------------------------------------
Beschreibung


-------------------------------------------------------------------------------
Input
-

Output
-
******************************************************************************)
METHOD PUBLIC Close : ERetCode_t
VAR_INPUT
END_VAR

	Close := ERetCode_t.eRetBusy;
	
	fbClose.hFile 		:= fbOpen.hFile;

	IF o_bEmpty = TRUE THEN

		fbClose.bExecute 	:= TRUE; 

		IF trgClose.Q = TRUE THEN
			o_bOpen 			:= FALSE;
		END_IF;	
		
		IF fbClose.bError = TRUE THEN
			Close := eRetCode_t.eRetFailed;
		END_IF;			

	END_IF;

	IF o_bOpen = FALSE THEN
		Close 				:= ERetCode_t.eRetDone;
		fbClose.bExecute 	:= FALSE;		
	END_IF;
END_METHOD

(******************************************************************************
Baustein: FB_TestReportBase.getFileName
Spezifikation: doc/Spezifikation.pdf, Kap. x.y.z
-------------------------------------------------------------------------------
erstellt:
von:
Geändert:
von:
-------------------------------------------------------------------------------
Beschreibung
Diese Methode muss vom ableitenden Baustein überschrieben werden und
wird von der Basisklasse aus aufgerufen wenn der Report erstellt werden
soll.

-------------------------------------------------------------------------------
Input
	i_pFileName : NameHandle_t;
	i_pPath		: PathHandle_t;

Output
-
******************************************************************************)
METHOD PROTECTED getFileName : ERetCode_t
VAR_INPUT
	i_pFileName : NameHandle_t;
	i_pPath		: PathHandle_t;
END_VAR
END_METHOD

(******************************************************************************
Baustein: FB_TestReportBase.getTime
Spezifikation: doc/Spezifikation.pdf, Kap. x.y.z
-------------------------------------------------------------------------------
erstellt:
von:
Geändert:
von:
-------------------------------------------------------------------------------
Beschreibung


-------------------------------------------------------------------------------
Input
-

Output
-
******************************************************************************)
METHOD PROTECTED getTime : TimeStruct
VAR_INPUT
END_VAR
VAR
END_VAR

	getTime := PRG_TestLib.getTime();
END_METHOD

(******************************************************************************
Baustein: FB_TestReportBase.Open
Spezifikation: doc/Spezifikation.pdf, Kap. x.y.z
-------------------------------------------------------------------------------
erstellt:
von:
Geändert:
von:
-------------------------------------------------------------------------------
Beschreibung


-------------------------------------------------------------------------------
Input
-

Output
-
******************************************************************************)
METHOD PUBLIC open : ERetCode_t
VAR_INPUT
	i_strPath : StrPathName_t;
	i_strName : StrFileName_t;
END_VAR

	open := ERetCode_t.eRetBusy;
	
	strFileName := i_strName;
	strFilePath := i_strPath;

	fbOpen.sPathName 	:= CONCAT(strFilePath, strFileName);
	fbOpen.nMode 	 	:= FOPEN_MODEWRITE OR FOPEN_MODEBINARY;	
	fbOpen.bExecute  	:= TRUE;
			
	IF trgOpen.Q = TRUE THEN
		o_bOpen := true;
		fbOpen.bExecute  := FALSE;		
	END_IF;	
	
	IF fbOpen.bError = TRUE THEN
		open := eRetCode_t.eRetFailed;
	END_IF;	

	IF o_bOpen = TRUE THEN
		open := eRetCode_t.eRetDone;
	END_IF;
END_METHOD

(******************************************************************************
Baustein: FB_TestReportBase.reset
Spezifikation: doc/Spezifikation.pdf, Kap. x.y.z
-------------------------------------------------------------------------------
erstellt:
von:
Geändert:
von:
-------------------------------------------------------------------------------
Beschreibung


-------------------------------------------------------------------------------
Input
-

Output
-
******************************************************************************)
METHOD PUBLIC reset : BOOL
VAR_INPUT
END_VAR

	IF fbOpen.hFile <> 0 THEN
		close();
	END_IF
	
	clearBuffer();

	fbOpen(sPathName := '', bExecute := FALSE);
	
	fbWrite(bExecute := FALSE);
	
	fbClose(bExecute := FALSE);
	
	o_bOpen := false;
END_METHOD

(******************************************************************************
Baustein: FB_TestReportBase.writeBuffer
Spezifikation: doc/Spezifikation.pdf, Kap. x.y.z
-------------------------------------------------------------------------------
erstellt:
von:
Geändert:
von:
-------------------------------------------------------------------------------
Beschreibung


-------------------------------------------------------------------------------
Input
-

Output
-
******************************************************************************)
METHOD PUBLIC writeBuffer : ERetCode_t
VAR_INPUT
END_VAR
VAR
	u32Len : UDINT;
END_VAR

	writeBuffer := eRetCode_t.eRetBusy;

	IF fbWrite.bBusy = TRUE THEN
		RETURN;	
	ELSIF u32WrIdx = u32RdIdx THEN
		writeBuffer := eRetCode_t.eRetDone;
		RETURN;	
	END_IF
	
	IF u32WrIdx > u32RdIdx THEN
		u32Len := u32WrIdx - u32RdIdx; 
		writeBuffer := writeData(i_pData := ADR(Buffer)+u32RdIdx, u32Size := u32Len);	
	ELSE
		u32Len := u32MaxIdx - u32RdIdx; 
		writeBuffer := writeData(i_pData := ADR(Buffer)+ u32RdIdx, u32Size := u32Len);
		writeBuffer := writeData(i_pData := ADR(Buffer), u32Size := u32WrIdx);	
	END_IF;
END_METHOD

(******************************************************************************
Baustein: FB_TestReportBase.writeData
Spezifikation: doc/Spezifikation.pdf, Kap. x.y.z
-------------------------------------------------------------------------------
erstellt:
von:
Geändert:
von:
-------------------------------------------------------------------------------
Beschreibung


-------------------------------------------------------------------------------
Input
	i_pData : POINTER TO BYTE;
	u32Size : UDINT;
	
Output
-
******************************************************************************)
METHOD PROTECTED writeData : ERetCode_t
VAR_INPUT
	i_pData : POINTER TO BYTE;
	u32Size : UDINT;
END_VAR

	writeData := ERetCode_t.eRetFailed;
	
	IF u32Size = 0 OR i_pData = 0 THEN
		RETURN;
	END_IF
	
	fbWrite.pWriteBuff 	:= i_pData; 
	fbWrite.cbWriteLen 	:= u32Size; 
	fbWrite.hFile 		:= fbOpen.hFile; 

	fbWrite(bExecute 	:= TRUE);
			
	IF fbWrite.bBusy = FALSE THEN
		fbWrite(bExecute 	:= FALSE);	
		writeData 	:= ERetCode_t.eRetDone;
		u32RdIdx 	:= u32WrIdx;
	ELSE	
		writeData := ERetCode_t.eRetBusy;
	END_IF;	

	IF fbWrite.bError = TRUE THEN
		writeData := eRetCode_t.eRetFailed;
	END_IF;
END_METHOD

END_FUNCTION_BLOCK

// ---- Source/Report/Format/FB_XmlTag.TcPOU
FUNCTION_BLOCK FB_XmlTag
IMPLEMENTS IFileData_t
VAR
	strBuffer 		: STRING(1024);
	strName   		: STRING;
	strTagEnd 		: STRING;
	u32Attributes 	: UDINT;
	strTags 			: STRING(1024);
	u32Tag 	      : UDINT;
	eFormat  		: EXmlFormat_t;
	strTemp 			: STRING(1024);
	u32Size 			: UDINT;
	strCRLF   		: STRING := '$R$N';
END_VAR

METHOD PUBLIC AddAttribute : Reference to FB_XmlTag
VAR_INPUT
	strName  : STRING;
	strValue : STRING;
END_VAR
VAR
	strAttr  : STRING(255);
END_VAR

	AddAttribute REF= THIS^;

	strAttr := ' ';
	strAttr := concat(strAttr, strName);
	strAttr := concat(strAttr, '="');
	strAttr := concat(strAttr, strValue);
	strAttr := concat(strAttr, '"');
	
	strBuffer := concat(strBuffer, strAttr);
	
	u32Attributes := u32Attributes+1;
	
	calculateSize();
END_METHOD

METHOD PUBLIC AddTag : BOOL
VAR_INPUT
	fbXml : FB_XmlTag;
END_VAR
VAR	
	strTag : STRING(1024);
END_VAR

	strTag 	 := fbXml.getXml();
	
	_CONCAT(ADR(strTags), SIZEOF(strTags), ADR(strTag), SIZEOF(strTag));
	
	u32Tag := u32Tag + 1;
		
	calculateSize();
END_METHOD

METHOD PRIVATE calculateSize

	u32Size := to_udint(len(strBuffer) + len(strTags));
END_METHOD

METHOD PUBLIC close : BOOL

	strBuffer := concat(strBuffer, '/>');
	
	IF eFormat = EXmlFormat_t.eStructuredXml THEN
		_CONCAT(ADR(strBuffer), SIZEOF(strBuffer), ADR(strCRLF), SIZEOF(strCRLF));
	END_IF	

	strTagEnd := '</';
	strTagEnd := CONCAT(strTagEnd, strName);
	strTagEnd := CONCAT(strTagEnd, '>');	
	
	IF eFormat = EXmlFormat_t.eStructuredXml THEN
		_CONCAT(ADR(strTagEnd), SIZEOF(strTagEnd), ADR(strCRLF), SIZEOF(strCRLF));
	END_IF
END_METHOD

METHOD PUBLIC create : reference to FB_XmlTag
VAR_INPUT
	strValue : STRING;
END_VAR

	create REF= THIS^;
	
	u32Attributes := 0;
	u32Tag        := 0;
	strName   	  := strValue;
	strTags 		  := '';
	strBuffer 	  := '<';
	strBuffer 	  := concat(strBuffer, strName);	
	

	
	calculateSize();
END_METHOD

METHOD getDataPtr : POINTER TO BYTE

	getXml();
	
	getDataPtr := adr(strTemp);
END_METHOD

METHOD getSize : UDINT

	getXml();

	getSize := _len(ADR(strTemp), SIZEOF(strTemp));
END_METHOD

METHOD PUBLIC getXml : STRING(1024)
VAR
	u32Len    : UDINT;	
END_VAR

	u32Len := _len(ADR(strBuffer), SIZEOF(strBuffer));

	MEMSET(ADR(strTemp), 0, SIZEOF(strTemp));

	_CONCAT(ADR(strTemp), SIZEOF(strTemp), ADR(strBuffer), SIZEOF(strBuffer));
			
	IF u32Tag > 0 THEN
		
		strTemp := DELETE(strTemp, 1, UDINT_TO_INT(u32Len-3));
						
		_CONCAT(ADR(strTemp), SIZEOF(strTemp), ADR(strTags), SIZEOF(strTags));
		
		_CONCAT(ADR(strTemp), SIZEOF(strTemp), ADR(strTagEnd), SIZEOF(strTagEnd));
		
	END_IF;
	
	getXml := strTemp;
END_METHOD

METHOD PUBLIC setFormat : REFERENCE TO FB_XmlTag
VAR_INPUT
	eFormat : EXmlFormat_t;
END_VAR

	setFormat REF= THIS^;
	
	this^.eFormat := eFormat;
END_METHOD

END_FUNCTION_BLOCK

// ---- Source/Report/Format/_CONCAT.TcPOU
FUNCTION _CONCAT : BOOL
VAR_INPUT
	pDst 	 		: POINTER TO BYTE;
	u32DstSize 	: UDINT;
	pSrc 	 		: POINTER TO BYTE;
	u32SrcSize 	: UDINT;
END_VAR
VAR
	u32DstLen 	: UDINT;
	u32SrcLen   : UDINT;
END_VAR


	_CONCAT := FALSE;
	u32SrcLen  := _LEN(pSrc, u32SrcSize);
	u32DstLen  := _LEN(pDst, u32DstSize);
				
	IF u32SrcLen + u32DstLen > (u32DstSize) THEN
		RETURN;
	END_IF
	
	pDst := pDst + u32DstLen;
	 
	MEMCPY(pDst, pSrc, u32SrcLen);
	
	pDst := pDst+u32SrcLen;
	
	pDst^ := 0;
	
	_CONCAT := TRUE;

END_FUNCTION

// ---- Source/Report/Format/_LEN.TcPOU
FUNCTION _LEN : UDINT
VAR_INPUT
	pSrc 	 : POINTER TO BYTE;
	u32Max : UDINT;
END_VAR

	
	_len := 0;

	WHILE (pSrc^ <> 0 and _len < u32Max) DO
		_len := _len+1;
		pSrc := pSrc+1;
	END_WHILE

END_FUNCTION

// ---- Test/PRG_Temp.TcPOU
PROGRAM PRG_Temp
VAR
	xmlTag	  	: FB_XmlTag;
	xmlPassed  	: FB_XmlTag;
	xmlFailed  	: FB_XmlTag;
	xmlSkipped 	: FB_XmlTag;
	bTest 		: BOOL;
	
	
	xmlTestsuites	  	: FB_XmlTag;
	xmlTestsuite	  	: FB_XmlTag;
	xmlTest	  			: FB_XmlTag;
	xmlTestResult		: FB_XmlTag;
	
	xml : STRING(255);

	a_iTestSuite 	: ARRAY [0..255] OF ITestSuite_t;
	u16TestSuites 	: UINT;
	u16Index	  	: UINT;
	iActTestSuite 	: ITestSuite_t;
	pTestReport		: POINTER TO FB_TestReportBase;
	eRetCode 		: ERetCode_t;

	fbSystemTime 	: FB_LocalSystemTime;
	
	fbUnittest 		: FB_CoverageFile;
	u16ReportState  : UINT;
	u16TestSuitIdx	: UINT;
	iTestCase  		: ITestBase_t;
	sTempResult     : SStatistic_t;
END_VAR


	IF bTest THEN
		btest := FALSE;
		xmlTag.create('Testcase')
			.AddAttribute('name', 			'Testid 1')
			.AddAttribute('assertions', 	'6')
			.AddAttribute('classname', 	'ctest')
			.AddAttribute('time', 			'0.100')
			.close();
			
		xmlPassed.create('passed').close();
		xmlFailed.create('failed').AddAttribute('message', 'quark').close();
		xmlSkipped.create('skipped').close();	
		
		xmlTag.AddTag(xmlFailed);
		
		
		xml := xmlTag.getXml();
		
	END_IF

END_PROGRAM

// ---- Source/Report/File/FB_TextReport.TcPOU
FUNCTION_BLOCK FB_TextReport EXTENDS FB_TestReportBase

(******************************************************************************
Baustein: FB_TestReportBase.BuildFile
Spezifikation: doc/Spezifikation.pdf, Kap. x.y.z
-------------------------------------------------------------------------------
erstellt:
von:
Geändert:
von:
-------------------------------------------------------------------------------
Beschreibung
Diese Methode muss vom ableitenden Baustein überschrieben werden und
wird von der Basisklasse aus aufgerufen wenn der Report erstellt werden
soll.

-------------------------------------------------------------------------------
Input
-

Output
-
******************************************************************************)
METHOD PROTECTED BuildFile : ERetCode_t
VAR_INPUT
	i_u32Line : UDINT;
END_VAR

	BuildFile := ERetCode_t.eRetBusy;

	CASE i_u32Line OF

	0: addString('Test Report :');
	   addDate(getTime());
	   addString(' - ');
	   addTime(getTime());
	1: addString('++++++++++++++++++++++++++++++++++++++++++++++++++');
	2: //
	3: //

	4: addString('Asserts gesamt: ');
	   addValue(sStatistic.u32Asserts);

	5: addString('Asserts passed: ');
	   addValue(sStatistic.u32Passed);

	6: addString('Asserts failed: ');
	   addValue(sStatistic.u32Failed);

	7: //

	9:  addString('Ergebnis : ');
		IF sStatistic.u32Failed > 0 THEN
			addString('FAILED');
		ELSE
			addString('PASSED');
		END_IF;

	10: addString('++++++++++++++++++++++++++++++++++++++++++++++++++');
	
	99: BuildFile := ERetCode_t.eRetDone;

	END_CASE;
END_METHOD

(******************************************************************************
Baustein: FB_TestReportBase.getFileName
Spezifikation: doc/Spezifikation.pdf, Kap. x.y.z
-------------------------------------------------------------------------------
erstellt:
von:
Geändert:
von:
-------------------------------------------------------------------------------
Beschreibung
Diese Methode muss vom ableitenden Baustein überschrieben werden und
wird von der Basisklasse aus aufgerufen wenn der Report erstellt werden
soll.

-------------------------------------------------------------------------------
Input
-

Output
-
******************************************************************************)
METHOD PROTECTED getFileName : ERetCode_t
VAR_INPUT
	i_pFileName : NameHandle_t;
	i_pPath		: PathHandle_t;
END_VAR
VAR
	sTime : TIMESTRUCT;
END_VAR

	i_pFileName^ := 'Exp_';
	i_pPath^ 	 := 'C:\Users\Administrator\Desktop\TestResult\';

	sTime := getTime();

	i_pFileName^ := Concat(i_pFileName^, WORD_TO_STRING(sTime.wYear));
	i_pFileName^ := Concat(i_pFileName^, DWORD_TO_DECSTR(sTime.wMonth, 2));
	i_pFileName^ := Concat(i_pFileName^, DWORD_TO_DECSTR(sTime.wDay  , 2));
	i_pFileName^ := Concat(i_pFileName^, '_');
	i_pFileName^ := Concat(i_pFileName^, DWORD_TO_DECSTR(sTime.wHour  , 2));
	i_pFileName^ := Concat(i_pFileName^, DWORD_TO_DECSTR(sTime.wMinute, 2));
	i_pFileName^ := Concat(i_pFileName^, '.txt');
END_METHOD

END_FUNCTION_BLOCK

// ---- Source/Testsuite/FB_Testsuite.TcPOU
(******************************************************************************
Baustein: FB_Testsuite
Spezifikation: doc/Spezifikation.pdf, Kap. x.y.z
-------------------------------------------------------------------------------
erstellt:
von:
Geändert:
von:
-------------------------------------------------------------------------------
Beschreibung
Dieser Baustein enthält alle zugeordneten Testfälle. Ein Testfall
ist ein abgeleiteter Baustein (FB) von FB_TestBase.

-------------------------------------------------------------------------------
Input
-

Output
-
******************************************************************************)
FUNCTION_BLOCK FB_Testsuite
IMPLEMENTS ITestsuite_t
VAR_OUTPUT
	o_eState  		: EState_t;
	o_eResult 		: EResult_t;
END_VAR
VAR
	strId				: ObjectId_t;
	strPath			: ObjectId_t;
	bRegistered    : BOOL;
	a_iTest  		: ARRAY [0..255] OF ITestBase_t;
	iTest     		: ITestBase_t;
	u16TestCases  	: UINT;
	u16Index 		: UINT;
	sStatistic 		: SStatistic_t;
END_VAR

(******************************************************************************
Baustein: FB_Testsuite.addTestcase
Spezifikation: doc/Spezifikation.pdf, Kap. x.y.z
-------------------------------------------------------------------------------
erstellt:
von:
Geändert:
von:
-------------------------------------------------------------------------------
Beschreibung
Diese Methode

-------------------------------------------------------------------------------
Input
i_pTestCase

Output
-
******************************************************************************)
{attribute 'hide'} 
METHOD PUBLIC addTestcase : BOOL
VAR_INPUT
	i_iTestCase : ITestBase_t;
END_VAR

	addTestcase := FALSE;

	IF 	i_iTestCase  <> 0   AND 
		u16TestCases <  255 THEN
		
		a_iTest[u16TestCases] := i_iTestCase;
		
		u16TestCases := u16TestCases +1;
		
		sStatistic.u32TestCases := sStatistic.u32TestCases + 1;
		
		addTestcase := true;
	END_IF
END_METHOD

METHOD execute : BOOL
VAR_INPUT
	i_bStart	: BOOL;
END_VAR
VAR
    sTestResult : STestcase_t;
END_VAR

	CASE o_eState OF
		
	EState_t.eStateInit:
	
		o_eState 	:= EState_t.eStateError;
		IF bRegistered = TRUE THEN
			o_eState 	:= EState_t.eStateIdle;
		END_IF;
		
	EState_t.eStateIdle:

		u16Index := 0;

		IF i_bStart = TRUE THEN
			logInfo(CONCAT('Run Testsuite ', strId));
			iTest 	 := getFirstTestCase();
			IF iTest <> 0 THEN
				logInfo(CONCAT('Execute Testcase ', iTest.getId()));
			END_IF;
			sStatistic.u32Executed  := 0;
			sStatistic.u32Passed 	:= 0;
			sStatistic.u32Failed 	:= 0;
			sStatistic.u32Asserts 	:= 0;
			o_eState  := EState_t.eStatePrepare;
			o_eResult := EResult_t.eStatePassed;
		END_IF;

	EState_t.eStatePrepare:

		IF iTest <> 0 THEN
			sTestResult := iTest.Result;
			IF sTestResult.eState <> EResult_t.eStateSkipped THEN
				 IF iTest._prepare() = ERetCode_t.eRetDone THEN
					  o_eState := EState_t.eStateExecute;
				 END_IF;
			ELSE
				 iTest 	:= getNextTestCase();
			END_IF;
		ELSE
			o_eState := EState_t.eStateREady;			
		END_IF;

	EState_t.eStateExecute:

		sTestResult := iTest.Result;

		IF iTest._execute()    = ERetCode_t.eRetDone		 	  OR 
			sTestResult.eState  = EResult_t.eStateFailedFatal THEN
			
			sStatistic.u32Executed := sStatistic.u32Executed + 1;	
			  (* update Result *)
			sTestResult := iTest.Result;
		
			sStatistic.u32Passed 	:= sStatistic.u32Passed + sTestResult.u32Passed;
			sStatistic.u32Failed 	:= sStatistic.u32Failed + sTestResult.u32Failed;
			sStatistic.u32Asserts   := sStatistic.u32Passed + sStatistic.u32Failed;
			
			// Status des aktuellen Tests auswerten
			CASE sTestResult.eState OF
			EResult_t.eStatePassed     : logInfo('	Test Passed');
			EResult_t.eStateFailed     : logInfo('	Test Failed');
			EResult_t.eStateFailedFatal: logInfo('	Test Failed Fatal');	
			END_CASE
			
			// Status der Testsuite ermitteln
			CASE o_eResult OF 

			EResult_t.eStatePassed:
				// Status des letzen Tests übernehmen
				o_eResult := sTestResult.eState;
				

			EResult_t.eStateFailed:
				// Status nur übernehmen wenn ein Fatal-Status
				// ermittelt wird und der Test sofort abgebrochen
				// werden soll.
				IF sTestResult.eState = EResult_t.eStateFailedFatal THEN
					o_eResult := sTestResult.eState;
					o_eState  := EState_t.eStateCleanUp;
				END_IF;		

			END_CASE;

			o_eState := EState_t.eStateCleanUp;

			IF o_eResult = EResult_t.eStateFailedFatal THEN
				o_eState := EState_t.eStateReady;					
			END_IF;

		END_IF;

	ESTate_t.eStateCleanUp:

		IF iTest <> 0 THEN
			IF iTest._cleanup() = ERetCode_t.eRetDone THEN
				iTest 	:= getNextTestCase();
				o_eState := EState_t.eStatePrepare;
			END_IF;
		ELSE
			o_eState := EState_t.eStateReady;
		END_IF;
		
	ESTate_t.eStateReady:
	
		IF i_bStart = FALSE THEN
			o_eState := EState_t.eStateIdle;
		END_IF
		
	ESTate_t.eStateError:	
		
		// wenn wir hier rauskommen ist was dummes passiert
		
	ELSE
		
		o_eState := EState_t.eStateError;
		
	END_CASE;
	
	
	
	
	
	
//
END_METHOD

(******************************************************************************
Baustein: FB_Testsuite.FB_init
Spezifikation: doc/Spezifikation.pdf, Kap. x.y.z
-------------------------------------------------------------------------------
erstellt:
von:
Geändert:
von:
-------------------------------------------------------------------------------
Beschreibung
Diese Methode

-------------------------------------------------------------------------------
Input
i_pTestCase

Output
-
******************************************************************************)
{attribute 'hide'} 
METHOD FB_init : BOOL
VAR_INPUT
	bInitRetains 	: BOOL; // if TRUE, the retain variables are initialized (warm start / cold start)
	bInCopyCode 	: BOOL;  // if TRUE, the instance afterwards gets moved into the copy code (online change)
	i_strId	  		: ObjectId_t;
	i_strPath		: ObjectId_t;
END_VAR

	strId 	:= i_StrId;
	strPath := i_strPath;
	register();
END_METHOD

(******************************************************************************
Baustein: FB_Testsuite.getFirstTestCase
Spezifikation: doc/Spezifikation.pdf, Kap. x.y.z
-------------------------------------------------------------------------------
erstellt:
von:
Geändert:
von:
-------------------------------------------------------------------------------
Beschreibung
Diese Methode

-------------------------------------------------------------------------------
Input
-

Output
-
******************************************************************************)
{attribute 'hide'} 
METHOD PUBLIC getFirstTestCase : ITestBase_t
VAR_INPUT
END_VAR

	u16Index := 0;
	getFirstTestCase := a_iTest[0];
END_METHOD

(******************************************************************************
Baustein: FB_Testsuite.getId
Spezifikation: doc/Spezifikation.pdf, Kap. x.y.z
-------------------------------------------------------------------------------
erstellt:
von:
Geändert:
von:
-------------------------------------------------------------------------------
Beschreibung
Diese Methode

-------------------------------------------------------------------------------
Input
-

Output
-
******************************************************************************)
{attribute 'hide'} 
METHOD PUBLIC getId : STRING
VAR_INPUT
END_VAR

	getId := strId;
END_METHOD

(******************************************************************************
Baustein: FB_Testsuite.getNextTestCase
Spezifikation: doc/Spezifikation.pdf, Kap. x.y.z
-------------------------------------------------------------------------------
erstellt:
von:
Geändert:
von:
-------------------------------------------------------------------------------
Beschreibung
Diese Methode

-------------------------------------------------------------------------------
Input
-

Output
-
******************************************************************************)
{attribute 'hide'} 
METHOD PUBLIC getNextTestCase : ITestBase_t
VAR_INPUT
END_VAR

	getNextTestCase := 0;
	u16Index 		 := u16Index + 1;

	IF u16Index < u16TestCases THEN
		getNextTestCase := a_iTest[u16Index];
	END_IF;
END_METHOD

{attribute 'hide'} 
METHOD PUBLIC getPath : ObjectId_t
VAR_INPUT
END_VAR

	getPath := strPath;
END_METHOD

METHOD getResult : EResult_t
VAR_INPUT
END_VAR

	getResult := o_eResult;
END_METHOD

METHOD getState : EState_t
getState := o_eState;
END_METHOD

(******************************************************************************
Baustein: FB_Testsuite.logInfo
Spezifikation: doc/Spezifikation.pdf, Kap. x.y.z
-------------------------------------------------------------------------------
erstellt:
von:
Geändert:
von:
-------------------------------------------------------------------------------
Beschreibung
Diese Methode

-------------------------------------------------------------------------------
Input
i_strMessage

Output
-
******************************************************************************)
{attribute 'hide'} 
METHOD PROTECTED logInfo : BOOL
VAR_INPUT
	i_strMessage : StrMessage_t;
END_VAR

	ADSLOGSTR(msgCtrlMask 	:= ADSLOG_MSGTYPE_HINT , 
			  msgFmtStr 	:= i_strMessage, 
			  strArg 		:= '');
END_METHOD

(******************************************************************************
Baustein: FB_Testsuite.register
Spezifikation: doc/Spezifikation.pdf, Kap. x.y.z
-------------------------------------------------------------------------------
erstellt:
von:
Geändert:
von:
-------------------------------------------------------------------------------
Beschreibung
Diese Methode

-------------------------------------------------------------------------------
Input
-

Output
-
******************************************************************************)
{attribute 'hide'} 
METHOD PROTECTED register : BOOL
VAR_INPUT
END_VAR

	bRegistered := PRG_TestLib.addTestSuite(this^);
END_METHOD

PROPERTY Result : SStatistic_t
GET
Result := sStatistic;
END_GET
END_PROPERTY

END_FUNCTION_BLOCK

// ---- Test/FB_Test_Base.TcPOU
{attribute 'hide'}
FUNCTION_BLOCK FB_Test_Base EXTENDS FB_TestBase

(******************************************************************************
Baustein: FB_Test_Base.cleanup
Spezifikation: doc/Spezifikation.pdf, Kap. x.y.z
-------------------------------------------------------------------------------
erstellt:
von:
Geändert:
von:
-------------------------------------------------------------------------------
Beschreibung
Diese Methode...

-------------------------------------------------------------------------------
Input
-

Output
-
******************************************************************************)
METHOD PUBLIC cleanup : ERetCode_t
VAR_INPUT
END_VAR

	cleanup := ERetCode_t.eRetDone;
END_METHOD

(******************************************************************************
Baustein: FB_Test_Base.execute
Spezifikation: doc/Spezifikation.pdf, Kap. x.y.z
-------------------------------------------------------------------------------
erstellt:
von:
Geändert:
von:
-------------------------------------------------------------------------------
Beschreibung
Diese Methode...

-------------------------------------------------------------------------------
Input
-

Output
-
******************************************************************************)
METHOD PUBLIC execute : ERetCode_t
VAR_INPUT
END_VAR
VAR
	bValue1   : ARRAY[0..10] OF BOOL;
	bValue2   : ARRAY[0..10] OF BOOL;
	s8Value1  : ARRAY[0..10] OF SINT;
	s8Value2  : ARRAY[0..10] OF SINT;
	u8Value1  : ARRAY[0..10] OF USINT;
	u8Value2  : ARRAY[0..10] OF USINT;	
	s16Value1 : ARRAY[0..10] OF INT;
	s16Value2 : ARRAY[0..10] OF INT;
	u16Value1 : ARRAY[0..10] OF UINT;
	u16Value2 : ARRAY[0..10] OF UINT;		
	s32Value1 : ARRAY[0..10] OF DINT;
	s32Value2 : ARRAY[0..10] OF DINT;
	u32Value1 : ARRAY[0..10] OF UDINT;
	u32Value2 : ARRAY[0..10] OF UDINT;	
	r32Value1 : ARRAY[0..10] OF REAL;
	r32Value2 : ARRAY[0..10] OF REAL;
	r64Value1 : ARRAY[0..10] OF LREAL;
	r64Value2 : ARRAY[0..10] OF LREAL;
	strValue1 : ARRAY[0..10] OF STRING;
	strValue2 : ARRAY[0..10] OF STRING;
END_VAR


	bValue1[0] := TRUE;
	bValue2[0] := TRUE;
	
	setMessage('Teste Datentyp BOOL');
	assert.EQUAL(bValue1[0], bValue2[0]);
	
	setMessage('Teste Datentyp Array of BOOL');
	assert.EQUAL(bValue1, bValue2);

(**********************************************) 
	
	s8Value1[0] := 32;
	s8Value2[0] := 32;
	
	setMessage('Teste Datentyp SINT');
	assert.EQUAL(s8Value1[0], s8Value2[0]);

	setMessage('Teste Datentyp Array of SINT');
	assert.EQUAL(s8Value1, s8Value2);
(**********************************************) 	

	u8Value1[0] := 34;
	u8Value2[0] := 34;
	
	setMessage('Teste Datentyp USINT');
	assert.EQUAL(u8Value1[0], u8Value2[0]);

	setMessage('Teste Datentyp Array of USINT');
	assert.EQUAL(u8Value1, u8Value2);
(**********************************************) 	
	
	s16Value1[0] := 1323;
	s16Value2[0] := 1323;
	
	setMessage('Teste Datentyp INT');
	assert.EQUAL(s16Value1[0], s16Value2[0]);

	setMessage('Teste Datentyp Array of INT');
	assert.EQUAL(s16Value1, s16Value2);
(**********************************************) 	

	u16Value1[0] := 3124;
	u16Value2[0] := 3124;
	
	setMessage('Teste Datentyp UINT');
	assert.EQUAL(u16Value1[0] , u16Value2[0] );

	setMessage('Teste Datentyp Array of UINT');
	assert.EQUAL(u16Value1 , u16Value2);
(**********************************************) 	

	s32Value1[0] := 1244;
	s32Value2[0] := 1244;
	
	setMessage('Teste Datentyp DINT');
	assert.EQUAL(s32Value1[0], s32Value2[0]);

	setMessage('Teste Datentyp Array of DINT');
	assert.EQUAL(s32Value1, s32Value2);
(**********************************************) 	

	u32Value1[0] := 4344;
	u32Value2[0] := 4344;
	
	setMessage('Teste Datentyp UDINT');
	assert.EQUAL(u32Value1[0], u32Value2[0]);

	setMessage('Teste Datentyp Array of UDINT');
	assert.EQUAL(u32Value1, u32Value2);
(**********************************************) 	

	r32Value1[0] := 133.53245;
	r32Value2[0] := 133.53245;
	
	setMessage('Teste Datentyp REAL');
	assert.EQUAL(r32Value1[0], r32Value2[0]);

	setMessage('Teste Datentyp Array of REAL');
	assert.EQUAL(r32Value1, r32Value2);
(**********************************************) 	

	r64Value1[0] := 1232.53325;
	r64Value2[0] := 1232.53325;

	setMessage('Teste Datentyp LREAL');
	assert.EQUAL(r64Value1[0], r64Value2[0]);

	setMessage('Teste Datentyp Array of LREAL');
	assert.EQUAL(r64Value1, r64Value2);

(**********************************************) 	

	strValue1[0] := 'Hallo Welt';
	strValue2[0] := 'Hallo Welt';

	setMessage('Teste Datentyp String ist gleich');
	assert.StringEqual(ADR(strValue1[0]), ADR(strValue2[0]));

	//setMessage('Teste Datentyp Array of String ist gleich');
	//assertEQUAL(strValue1, strValue2);

	strValue1[0] := 'Hallo Well';
	strValue2[0] := 'Hallo Welt';
	
	setMessage('Teste Datentyp String ist ungleich');
	assert.StringNotEqual(ADR(strValue1[0]), ADR(strValue2[0]));

	//setMessage('Teste Datentyp Array of String ist ungleich');
	//assert.NotEQUAL(strValue1, strValue2);
	
(**********************************************) 	





	execute := ERetCode_t.eRetDone;
END_METHOD

(******************************************************************************
Baustein: FB_Test_Base.prepare
Spezifikation: doc/Spezifikation.pdf, Kap. x.y.z
-------------------------------------------------------------------------------
erstellt:
von:
Geändert:
von:
-------------------------------------------------------------------------------
Beschreibung
Diese Methode...

-------------------------------------------------------------------------------
Input
-

Output
-
******************************************************************************)
METHOD PUBLIC prepare : ERetCode_t
VAR_INPUT
END_VAR

	prepare := ERetCode_t.eRetDone;
END_METHOD

END_FUNCTION_BLOCK

// ---- Test/FB_Test_Base_Ptr.TcPOU
{attribute 'hide'}
FUNCTION_BLOCK FB_Test_Base_Ptr EXTENDS FB_TestBase

(******************************************************************************
Baustein: FB_Test_Base.cleanup
Spezifikation: doc/Spezifikation.pdf, Kap. x.y.z
-------------------------------------------------------------------------------
erstellt:
von:
Geändert:
von:
-------------------------------------------------------------------------------
Beschreibung
Diese Methode...

-------------------------------------------------------------------------------
Input
-

Output
-
******************************************************************************)
METHOD PUBLIC cleanup : ERetCode_t
VAR_INPUT
END_VAR

	cleanup := ERetCode_t.eRetDone;
END_METHOD

(******************************************************************************
Baustein: FB_Test_Base.execute
Spezifikation: doc/Spezifikation.pdf, Kap. x.y.z
-------------------------------------------------------------------------------
erstellt:
von:
Geändert:
von:
-------------------------------------------------------------------------------
Beschreibung
Diese Methode...

-------------------------------------------------------------------------------
Input
-

Output
-
******************************************************************************)
METHOD PUBLIC execute : ERetCode_t
VAR_INPUT
END_VAR
VAR
	bValue1   : ARRAY[0..10] OF BOOL;
	bValue2   : ARRAY[0..10] OF BOOL;
	s8Value1  : ARRAY[0..10] OF SINT;
	s8Value2  : ARRAY[0..10] OF SINT;
	u8Value1  : ARRAY[0..10] OF USINT;
	u8Value2  : ARRAY[0..10] OF USINT;	
	s16Value1 : ARRAY[0..10] OF INT;
	s16Value2 : ARRAY[0..10] OF INT;
	u16Value1 : ARRAY[0..10] OF UINT;
	u16Value2 : ARRAY[0..10] OF UINT;		
	s32Value1 : ARRAY[0..10] OF DINT;
	s32Value2 : ARRAY[0..10] OF DINT;
	u32Value1 : ARRAY[0..10] OF UDINT;
	u32Value2 : ARRAY[0..10] OF UDINT;	
	r32Value1 : ARRAY[0..10] OF REAL;
	r32Value2 : ARRAY[0..10] OF REAL;
	r64Value1 : ARRAY[0..10] OF LREAL;
	r64Value2 : ARRAY[0..10] OF LREAL;
END_VAR


	bValue1[0] := TRUE;
	bValue2[0] := TRUE;
	
	setMessage('Teste Pointer to BOOL equal');
	assert.PtrEQUAL(ADR(bValue1[0]), ADR(bValue1[0]));
	
	setMessage('Teste Pointer to BOOL NOT equal');
	assert.PtrNOTEQUAL(ADR(bValue1), ADR(bValue2));

(**********************************************) 
	
	s8Value1[0] := 32;
	s8Value2[0] := 32;
	
	setMessage('Teste Pointer to BOOL SINT equal');
	assert.PtrEQUAL(ADR(s8Value1[0]), ADR(s8Value1[0]));

	setMessage('Teste Pointer to SINT not equal');
	assert.PtrNOTEQUAL(ADR(s8Value1), ADR(s8Value2));
(**********************************************) 	

	u8Value1[0] := 34;
	u8Value2[0] := 34;
	
	setMessage('Teste Pointer to USINT equal');
	assert.PtrEQUAL(ADR(u8Value1[0]), ADR(u8Value1[0]));

	setMessage('Teste Pointer to USINT not equal');
	assert.PtrNOTEQUAL(ADR(u8Value1), ADR(u8Value2));
(**********************************************) 	
	
	s16Value1[0] := 1323;
	s16Value2[0] := 1323;
	
	setMessage('Teste Pointer to INT equal');
	assert.PtrEQUAL(ADR(s16Value1[0]), ADR(s16Value1[0]));

	setMessage('Teste Pointer to INT not equal');
	assert.PtrNOTEQUAL(ADR(s16Value1), ADR(s16Value2));
(**********************************************) 	

	u16Value1[0] := 3124;
	u16Value2[0] := 3124;
	
	setMessage('Teste Pointer to UINT equal');
	assert.PtrEQUAL(ADR(u16Value1[0]) , ADR(u16Value1[0]) );

	setMessage('Teste Pointer to  UINT not equal');
	assert.PtrNOTEQUAL(ADR(u16Value1) , ADR(u16Value2));
(**********************************************) 	

	s32Value1[0] := 1244;
	s32Value2[0] := 1244;
	
	setMessage('Teste Pointer to DINT equal');
	assert.PtrEQUAL(ADR(s32Value1[0]), ADR(s32Value1[0]));

	setMessage('Teste Pointer to  DINT not equal');
	assert.PtrNOTEQUAL(ADR(s32Value1), ADR(s32Value2));
(**********************************************) 	

	u32Value1[0] := 4344;
	u32Value2[0] := 4344;
	
	setMessage('Teste Pointer to UDINT equal');
	assert.PtrEQUAL(ADR(u32Value1[0]), ADR(u32Value1[0]));

	setMessage('Teste Pointer to  UDINT not equal');
	assert.PtrNOTEQUAL(ADR(u32Value1), ADR(u32Value2));
(**********************************************) 	

	r32Value1[0] := 133.53245;
	r32Value2[0] := 133.53245;
	
	setMessage('Teste Pointer to REAL equal');
	assert.PtrEQUAL(ADR(r32Value1[0]), ADR(r32Value1[0]));

	setMessage('Teste Pointer to  REAL not equal');
	assert.PtrNOTEQUAL(ADR(r32Value1), ADR(r32Value2));
(**********************************************) 	

	r64Value1[0] := 1232.53325;
	r64Value2[0] := 1232.53325;

	setMessage('Teste Pointer to LREAL equal');
	assert.PtrEQUAL(ADR(r64Value1[0]), ADR(r64Value1[0]));

	setMessage('Teste Pointer to LREAL not equal');
	assert.PtrNOTEQUAL(ADR(r64Value1), ADR(r64Value2));

(**********************************************)

	setMessage('Teste Pointer = 0');	
	assert.PtrNull(pActual := 0);
	
	setMessage('Teste Pointer <> 0');	
	assert.PtrNotNull(pActual := ADR(r32Value1[0]));	
	
(**********************************************)	
	
	
	
	
	
	
	
	
	
	execute := ERetCode_t.eRetDone;
END_METHOD

(******************************************************************************
Baustein: FB_Test_Base.prepare
Spezifikation: doc/Spezifikation.pdf, Kap. x.y.z
-------------------------------------------------------------------------------
erstellt:
von:
Geändert:
von:
-------------------------------------------------------------------------------
Beschreibung
Diese Methode...

-------------------------------------------------------------------------------
Input
-

Output
-
******************************************************************************)
METHOD PUBLIC prepare : ERetCode_t
VAR_INPUT
END_VAR

	prepare := ERetCode_t.eRetDone;
END_METHOD

END_FUNCTION_BLOCK

// ---- Test/FB_Test_Base_Not.TcPOU
{attribute 'hide'}
FUNCTION_BLOCK FB_Test_Base_Not EXTENDS FB_TestBase

(******************************************************************************
Baustein: FB_Test_Base_Not.cleanup
Spezifikation: doc/Spezifikation.pdf, Kap. x.y.z
-------------------------------------------------------------------------------
erstellt:
von:
Geändert:
von:
-------------------------------------------------------------------------------
Beschreibung
Diese Methode...

-------------------------------------------------------------------------------
Input
-

Output
-
******************************************************************************)
METHOD PUBLIC cleanup : ERetCode_t
VAR_INPUT
END_VAR

	cleanup := ERetCode_t.eRetDone;
END_METHOD

(******************************************************************************
Baustein: FB_Test_Base_Not.execute
Spezifikation: doc/Spezifikation.pdf, Kap. x.y.z
-------------------------------------------------------------------------------
erstellt:
von:
Geändert:
von:
-------------------------------------------------------------------------------
Beschreibung
Diese Methode...

-------------------------------------------------------------------------------
Input
-

Output
-
******************************************************************************)
METHOD PUBLIC execute : ERetCode_t
VAR_INPUT
END_VAR
VAR
	bValue1   : ARRAY[0..10] OF BOOL;
	bValue2   : ARRAY[0..10] OF BOOL;
	s8Value1  : ARRAY[0..10] OF SINT;
	s8Value2  : ARRAY[0..10] OF SINT;
	u8Value1  : ARRAY[0..10] OF USINT;
	u8Value2  : ARRAY[0..10] OF USINT;	
	s16Value1 : ARRAY[0..10] OF INT;
	s16Value2 : ARRAY[0..10] OF INT;
	u16Value1 : ARRAY[0..10] OF UINT;
	u16Value2 : ARRAY[0..10] OF UINT;		
	s32Value1 : ARRAY[0..10] OF DINT;
	s32Value2 : ARRAY[0..10] OF DINT;
	u32Value1 : ARRAY[0..10] OF UDINT;
	u32Value2 : ARRAY[0..10] OF UDINT;	
	r32Value1 : ARRAY[0..10] OF REAL;
	r32Value2 : ARRAY[0..10] OF REAL;
	r64Value1 : ARRAY[0..10] OF LREAL;
	r64Value2 : ARRAY[0..10] OF LREAL;
END_VAR


	bValue1[0] := FALSE;
	bValue2[0] := TRUE;
	
	setMessage('Teste Datentyp BOOL');
	assert.NotEQUAL(bValue1[0], bValue2[0]);
	
	setMessage('Teste Datentyp Array of BOOL');
	assert.NotEQUAL(bValue1, bValue2);

(**********************************************) 
	
	s8Value1[0] := 31;
	s8Value2[0] := 32;
	
	setMessage('Teste Datentyp SINT');
	assert.NotEQUAL(s8Value1[0], s8Value2[0]);

	setMessage('Teste Datentyp Array SINT');
	assert.NotEQUAL(s8Value1, s8Value2);
(**********************************************) 	

	u8Value1[0] := 1;
	u8Value2[0] := 34;
	
	setMessage('Teste Datentyp USINT');
	assert.NotEQUAL(u8Value1[0], u8Value2[0]);

	setMessage('Teste Datentyp Array of USINT');
	assert.NotEQUAL(u8Value1, u8Value2);
(**********************************************) 	
	
	s16Value1[0] := 1323;
	s16Value2[0] := 4324;
	
	setMessage('Teste Datentyp INT');
	assert.NotEQUAL(s16Value1[0], s16Value2[0]);

	setMessage('Teste Datentyp Array of INT');
	assert.NotEQUAL(s16Value1, s16Value2);
(**********************************************) 	

	u16Value1[0] := 3124;
	u16Value2[0] := 4232;
	
	setMessage('Teste Datentyp UINT');
	assert.NotEQUAL(u16Value1[0] , u16Value2[0] );

	setMessage('Teste Datentyp Array of UINT');
	assert.NotEQUAL(u16Value1 , u16Value2);
(**********************************************) 	

	s32Value1[0] := 1244;
	s32Value2[0] := 1593;
	
	setMessage('Teste Datentyp DINT');
	assert.NotEQUAL(s32Value1[0], s32Value2[0]);

	setMessage('Teste Datentyp Array of DINT');
	assert.NotEQUAL(s32Value1, s32Value2);
(**********************************************) 	

	u32Value1[0] := 4344;
	u32Value2[0] := 3424;
	
	setMessage('Teste Datentyp UDINT');
	assert.NotEQUAL(u32Value1[0], u32Value2[0]);

	setMessage('Teste Datentyp Array of UDINT');
	assert.NotEQUAL(u32Value1, u32Value2);
(**********************************************) 	

	r32Value1[0] := 133.53245;
	r32Value2[0] := 5345.53245;
	
	setMessage('Teste Datentyp REAL');
	assert.NotEQUAL(r32Value1[0], r32Value2[0]);

	setMessage('Teste Datentyp Array of REAL');
	assert.NotEQUAL(r32Value1, r32Value2);
(**********************************************) 	

	r64Value1[0] := 1232.53325;
	r64Value2[0] := 1345.53325;

	setMessage('Teste Datentyp LREAL');
	assert.NotEQUAL(r64Value1[0], r64Value2[0]);

	setMessage('Teste Datentyp Array of LREAL');
	assert.NotEQUAL(r64Value1, r64Value2);

(**********************************************) 		
	execute := ERetCode_t.eRetDone;
END_METHOD

(******************************************************************************
Baustein: FB_Test_Base_Not.prepare
Spezifikation: doc/Spezifikation.pdf, Kap. x.y.z
-------------------------------------------------------------------------------
erstellt:
von:
Geändert:
von:
-------------------------------------------------------------------------------
Beschreibung
Diese Methode...

-------------------------------------------------------------------------------
Input
-

Output
-
******************************************************************************)
METHOD PUBLIC prepare : ERetCode_t
VAR_INPUT
END_VAR

	prepare := ERetCode_t.eRetDone;
END_METHOD

END_FUNCTION_BLOCK

// ---- Test/FB_Test_Base_Delay.TcPOU
{attribute 'hide'}
FUNCTION_BLOCK FB_Test_Base_Delay EXTENDS FB_TestBase
VAR
	fbDelay : TON;
END_VAR

(******************************************************************************
Baustein: FB_Test_Base_Delay.cleanup
Spezifikation: doc/Spezifikation.pdf, Kap. x.y.z
-------------------------------------------------------------------------------
erstellt:
von:
Geändert:
von:
-------------------------------------------------------------------------------
Beschreibung
Diese Methode...

-------------------------------------------------------------------------------
Input
-

Output
-
******************************************************************************)
METHOD PUBLIC cleanup : ERetCode_t
VAR_INPUT
END_VAR

	cleanup := ERetCode_t.eRetDone;
	
	fbDelay(IN := false);
END_METHOD

(******************************************************************************
Baustein: FB_Test_Base_Delay.execute
Spezifikation: doc/Spezifikation.pdf, Kap. x.y.z
-------------------------------------------------------------------------------
erstellt:
von:
Geändert:
von:
-------------------------------------------------------------------------------
Beschreibung
Diese Methode...

-------------------------------------------------------------------------------
Input
-

Output
-
******************************************************************************)
METHOD PUBLIC execute : ERetCode_t
VAR_INPUT
END_VAR
VAR
	bValue1  : BOOL;
	bValue2  : BOOL;
	s32Value1 : DINT;
	s32Value2 : DINT;
	r32Value1 : REAL;
	r32Value2 : REAL;
END_VAR

	fbDelay(PT := t#250ms);
	execute 	  := ERetCode_t.eRetBusy;

	bValue1 := TRUE;
	bValue2 := TRUE;
	assert.EQUAL(bValue1, bValue2);

	s32Value1 := 1593;
	s32Value2 := 1593;
	assert.EQUAL(s32Value1, s32Value2);

	r32Value1 := 5345.53245;
	r32Value2 := 5345.53245;
	assert.EQUAL(r32Value1, r32Value2);

	if fbDelay.Q then
		execute := ERetCode_t.eRetDone;
	end_if;
END_METHOD

(******************************************************************************
Baustein: FB_Test_Base_Delay.prepare
Spezifikation: doc/Spezifikation.pdf, Kap. x.y.z
-------------------------------------------------------------------------------
erstellt:
von:
Geändert:
von:
-------------------------------------------------------------------------------
Beschreibung
Diese Methode...

-------------------------------------------------------------------------------
Input
-

Output
-
******************************************************************************)
METHOD PUBLIC prepare : ERetCode_t
VAR_INPUT
END_VAR

	prepare := ERetCode_t.eRetDone;
	
	fbDelay.IN := true;
END_METHOD

END_FUNCTION_BLOCK
